LIN {X 0,Y 696.84,Z 1074.1,A -85,B 0,C 180,E1 3614.763,E2 3614.763} C_VEL
LIN {X 0,Y 697.033,Z 1060.691,A -85,B 0,C 180,E1 3616.923,E2 3616.923} C_VEL
LIN {X 0,Y 697.324,Z 1042.875,A -85,B 0,C 180,E1 3618.806,E2 3618.806} C_VEL
LIN {X 0,Y 697.62,Z 1019.345,A -85,B 0,C 180,E1 3620.491,E2 3620.491} C_VEL
LIN {X 0,Y 698.013,Z 992.248,A -85,B 0,C 180,E1 3621.752,E2 3621.752} C_VEL
LIN {X 0,Y 698.325,Z 962.562,A -85,B 0,C 180,E1 3622.528,E2 3622.528} C_VEL
LIN {X 0,Y 697.391,Z 928.875,A -85,B 0,C 180,E1 3622.939,E2 3622.939} C_VEL
LIN {X 0,Y 696.362,Z 923.03,A -85,B 0,C 180,E1 3623.04,E2 3623.04} C_VEL
LIN {X 0,Y 696.127,Z 923.03,A -85,B 0,C 180,E1 3627.121,E2 3627.121} C_VEL
LIN {X 0,Y 696.052,Z 923.03,A -85,B 0,C 180,E1 3632.136,E2 3632.136} C_VEL
LIN {X 0,Y 696.075,Z 923.03,A -85,B 0,C 180,E1 3637.436,E2 3637.436} C_VEL
LIN {X 0,Y 695.88,Z 923.03,A -85,B 0,C 180,E1 3642.402,E2 3642.402} C_VEL
LIN {X 0,Y 696.007,Z 923.03,A -85,B 0,C 180,E1 3647.688,E2 3647.688} C_VEL
LIN {X 0,Y 696.066,Z 923.03,A -85,B 0,C 180,E1 3652.556,E2 3652.556} C_VEL
LIN {X 0,Y 696.017,Z 923.03,A -85,B 0,C 180,E1 3657.859,E2 3657.859} C_VEL
LIN {X 0,Y 696.298,Z 923.03,A -85,B 0,C 180,E1 3662.878,E2 3662.878} C_VEL
LIN {X 0,Y 696.247,Z 923.03,A -85,B 0,C 180,E1 3668.339,E2 3668.339} C_VEL
LIN {X 0,Y 696.266,Z 923.03,A -85,B 0,C 180,E1 3673.602,E2 3673.602} C_VEL
LIN {X 0,Y 696.358,Z 923.03,A -85,B 0,C 180,E1 3678.728,E2 3678.728} C_VEL
LIN {X 0,Y 696.496,Z 923.03,A -85,B 0,C 180,E1 3683.762,E2 3683.762} C_VEL
LIN {X 0,Y 696.447,Z 923.03,A -85,B 0,C 180,E1 3688.746,E2 3688.746} C_VEL
LIN {X 0,Y 696.437,Z 923.03,A -85,B 0,C 180,E1 3692.476,E2 3692.476} C_VEL
LIN {X 0,Y 696.418,Z 923.03,A -85,B 0,C 180,E1 3696.217,E2 3696.217} C_VEL
LIN {X 0,Y 696.336,Z 923.03,A -85,B 0,C 180,E1 3701.25,E2 3701.25} C_VEL
LIN {X 0,Y 696.388,Z 923.03,A -85,B 0,C 180,E1 3706.372,E2 3706.372} C_VEL
LIN {X 0,Y 696.229,Z 923.03,A -85,B 0,C 180,E1 3711.638,E2 3711.638} C_VEL
LIN {X 0,Y 696.274,Z 923.03,A -85,B 0,C 180,E1 3715.71,E2 3715.71} C_VEL
LIN {X 0,Y 696.189,Z 923.03,A -85,B 0,C 180,E1 3719.933,E2 3719.933} C_VEL
LIN {X 0,Y 696.124,Z 923.03,A -85,B 0,C 180,E1 3724.422,E2 3724.422} C_VEL
LIN {X 0,Y 696.016,Z 923.03,A -85,B 0,C 180,E1 3729.003,E2 3729.003} C_VEL
LIN {X 0,Y 696.257,Z 923.03,A -85,B 0,C 180,E1 3734.256,E2 3734.256} C_VEL
LIN {X 0,Y 696.094,Z 923.03,A -85,B 0,C 180,E1 3739.422,E2 3739.422} C_VEL
LIN {X 0,Y 696.038,Z 923.03,A -85,B 0,C 180,E1 3744.113,E2 3744.113} C_VEL
LIN {X 0,Y 696.066,Z 923.03,A -85,B 0,C 180,E1 3748.598,E2 3748.598} C_VEL
LIN {X 0,Y 696.27,Z 923.03,A -85,B 0,C 180,E1 3752.885,E2 3752.885} C_VEL
LIN {X 0,Y 696.419,Z 923.03,A -85,B 0,C 180,E1 3755.045,E2 3755.045} C_VEL
LIN {X 0,Y 702.161,Z 942.704,A -85,B 0,C 180,E1 3755.601,E2 3755.601} C_VEL
LIN {X 0,Y 701.459,Z 983.403,A -85,B 0,C 180,E1 3756.655,E2 3756.655} C_VEL
LIN {X 0,Y 700.459,Z 1020.42,A -85,B 0,C 180,E1 3758.118,E2 3758.118} C_VEL
LIN {X 0,Y 699.341,Z 1055.77,A -85,B 0,C 180,E1 3760.059,E2 3760.059} C_VEL
LIN {X 0,Y 698.44,Z 1087.21,A -85,B 0,C 180,E1 3762.367,E2 3762.367} C_VEL
LIN {X 0,Y 697.692,Z 1115.392,A -85,B 0,C 180,E1 3765.095,E2 3765.095} C_VEL
LIN {X 0,Y 697.113,Z 1138.714,A -85,B 0,C 180,E1 3768.115,E2 3768.115} C_VEL
LIN {X 0,Y 696.808,Z 1156.179,A -85,B 0,C 180,E1 3771.267,E2 3771.267} C_VEL
LIN {X 0,Y 696.688,Z 1167.713,A -85,B 0,C 180,E1 3774.397,E2 3774.397} C_VEL
LIN {X 0,Y 696.627,Z 1173.967,A -85,B 0,C 180,E1 3777.512,E2 3777.512} C_VEL
LIN {X 0,Y 696.49,Z 1175.495,A -85,B 0,C 180,E1 3779.999,E2 3779.999} C_VEL
LIN {X 0,Y 696.656,Z 1173.847,A -85,B 0,C 180,E1 3782.485,E2 3782.485} C_VEL
LIN {X 0,Y 696.704,Z 1167.444,A -85,B 0,C 180,E1 3785.6,E2 3785.6} C_VEL
LIN {X 0,Y 696.77,Z 1155.784,A -85,B 0,C 180,E1 3788.73,E2 3788.73} C_VEL
LIN {X 0,Y 697.098,Z 1138.122,A -85,B 0,C 180,E1 3791.883,E2 3791.883} C_VEL
LIN {X 0,Y 697.634,Z 1114.595,A -85,B 0,C 180,E1 3794.904,E2 3794.904} C_VEL
LIN {X 0,Y 697.968,Z 1103.957,A -85,B 0,C 180,E1 3796.014,E2 3796.014} C_VEL
LIN {X 0,Y 694.387,Z 1093.241,A -85,B 0,C 180,E1 3797.118,E2 3797.118} C_VEL
LIN {X 0,Y 690.934,Z 1081.896,A -85,B 0,C 180,E1 3798.188,E2 3798.188} C_VEL
LIN {X 0,Y 692.119,Z 1048.543,A -85,B 0,C 180,E1 3800.528,E2 3800.528} C_VEL
LIN {X 0,Y 693.322,Z 1012.284,A -85,B 0,C 180,E1 3802.409,E2 3802.409} C_VEL
LIN {X 0,Y 694.361,Z 974.431,A -85,B 0,C 180,E1 3803.796,E2 3803.796} C_VEL
LIN {X 0,Y 694.245,Z 940.568,A -85,B 0,C 180,E1 3804.648,E2 3804.648} C_VEL
LIN {X 0,Y 688.268,Z 923.03,A -85,B 0,C 180,E1 3805.177,E2 3805.177} C_VEL
LIN {X 0,Y 688.234,Z 923.03,A -85,B 0,C 180,E1 3810.329,E2 3810.329} C_VEL
LIN {X 0,Y 688.148,Z 923.03,A -85,B 0,C 180,E1 3815.688,E2 3815.688} C_VEL
LIN {X 0,Y 688.036,Z 923.03,A -85,B 0,C 180,E1 3821.212,E2 3821.212} C_VEL
LIN {X 0,Y 688.049,Z 923.03,A -85,B 0,C 180,E1 3826.446,E2 3826.446} C_VEL
LIN {X 0,Y 688.208,Z 923.03,A -85,B 0,C 180,E1 3832.225,E2 3832.225} C_VEL
LIN {X 0,Y 688.212,Z 923.03,A -85,B 0,C 180,E1 3836.724,E2 3836.724} C_VEL
LIN {X 0,Y 688.234,Z 923.03,A -85,B 0,C 180,E1 3841.429,E2 3841.429} C_VEL
LIN {X 0,Y 688.093,Z 923.327,A -85,B 0,C 180,E1 3844.092,E2 3844.092} C_VEL
LIN {X 0,Y 695.508,Z 945.947,A -85,B 0,C 180,E1 3844.641,E2 3844.641} C_VEL
LIN {X 0,Y 695.052,Z 1003.247,A -85,B 0,C 180,E1 3845.392,E2 3845.392} C_VEL
LIN {X 0,Y 694.208,Z 1042.654,A -85,B 0,C 180,E1 3846.416,E2 3846.416} C_VEL
LIN {X 0,Y 693.113,Z 1079.521,A -85,B 0,C 180,E1 3847.875,E2 3847.875} C_VEL
LIN {X 0,Y 691.948,Z 1114.634,A -85,B 0,C 180,E1 3849.81,E2 3849.81} C_VEL
LIN {X 0,Y 690.803,Z 1145.44,A -85,B 0,C 180,E1 3852.063,E2 3852.063} C_VEL
LIN {X 0,Y 689.951,Z 1172.229,A -85,B 0,C 180,E1 3854.62,E2 3854.62} C_VEL
LIN {X 0,Y 689.296,Z 1195.231,A -85,B 0,C 180,E1 3857.51,E2 3857.51} C_VEL
LIN {X 0,Y 688.941,Z 1212.25,A -85,B 0,C 180,E1 3860.393,E2 3860.393} C_VEL
LIN {X 0,Y 688.809,Z 1224.727,A -85,B 0,C 180,E1 3863.398,E2 3863.398} C_VEL
LIN {X 0,Y 688.734,Z 1231.97,A -85,B 0,C 180,E1 3866.237,E2 3866.237} C_VEL
LIN {X 0,Y 688.725,Z 1235.095,A -85,B 0,C 180,E1 3868.754,E2 3868.754} C_VEL
LIN {X 0,Y 688.851,Z 1235.078,A -85,B 0,C 180,E1 3871.268,E2 3871.268} C_VEL
LIN {X 0,Y 688.802,Z 1230.721,A -85,B 0,C 180,E1 3874.414,E2 3874.414} C_VEL
LIN {X 0,Y 688.94,Z 1219.976,A -85,B 0,C 180,E1 3877.89,E2 3877.89} C_VEL
LIN {X 0,Y 689.179,Z 1204.28,A -85,B 0,C 180,E1 3881.071,E2 3881.071} C_VEL
LIN {X 0,Y 689.655,Z 1183.093,A -85,B 0,C 180,E1 3884.119,E2 3884.119} C_VEL
LIN {X 0,Y 690.437,Z 1157.494,A -85,B 0,C 180,E1 3886.867,E2 3886.867} C_VEL
LIN {X 0,Y 691.422,Z 1128.305,A -85,B 0,C 180,E1 3889.265,E2 3889.265} C_VEL
LIN {X 0,Y 692.587,Z 1094.665,A -85,B 0,C 180,E1 3891.361,E2 3891.361} C_VEL
LIN {X 0,Y 693.775,Z 1058.061,A -85,B 0,C 180,E1 3893.036,E2 3893.036} C_VEL
LIN {X 0,Y 694.758,Z 1021.242,A -85,B 0,C 180,E1 3894.199,E2 3894.199} C_VEL
LIN {X 0,Y 695.371,Z 982.472,A -85,B 0,C 180,E1 3894.941,E2 3894.941} C_VEL
LIN {X 0,Y 694.761,Z 941.711,A -85,B 0,C 180,E1 3895.435,E2 3895.435} C_VEL
LIN {X 0,Y 688.099,Z 923.03,A -85,B 0,C 180,E1 3895.984,E2 3895.984} C_VEL
LIN {X 0,Y 688.244,Z 923.03,A -85,B 0,C 180,E1 3901.101,E2 3901.101} C_VEL
LIN {X 0,Y 688.201,Z 923.03,A -85,B 0,C 180,E1 3906.369,E2 3906.369} C_VEL
LIN {X 0,Y 688.063,Z 923.03,A -85,B 0,C 180,E1 3911.697,E2 3911.697} C_VEL
LIN {X 0,Y 688.076,Z 923.03,A -85,B 0,C 180,E1 3917.096,E2 3917.096} C_VEL
LIN {X 0,Y 688.182,Z 923.03,A -85,B 0,C 180,E1 3922.242,E2 3922.242} C_VEL
LIN {X 0,Y 688.174,Z 923.03,A -85,B 0,C 180,E1 3926.707,E2 3926.707} C_VEL
LIN {X 0,Y 688.271,Z 923.03,A -85,B 0,C 180,E1 3931.439,E2 3931.439} C_VEL
LIN {X 0,Y 688.328,Z 923.03,A -85,B 0,C 180,E1 3936.726,E2 3936.726} C_VEL
LIN {X 0,Y 688.194,Z 923.03,A -85,B 0,C 180,E1 3940.782,E2 3940.782} C_VEL
LIN {X 0,Y 688.276,Z 923.03,A -85,B 0,C 180,E1 3946.026,E2 3946.026} C_VEL
LIN {X 0,Y 688.465,Z 923.03,A -85,B 0,C 180,E1 3951.163,E2 3951.163} C_VEL
LIN {X 0,Y 688.379,Z 923.03,A -85,B 0,C 180,E1 3956.225,E2 3956.225} C_VEL
LIN {X 0,Y 688.46,Z 923.03,A -85,B 0,C 180,E1 3956.751,E2 3956.751} C_VEL
LIN {X 0,Y 690.605,Z 940.887,A -85,B 0,C 180,E1 3956.98,E2 3956.98} C_VEL
LIN {X 0,Y 690.561,Z 973.087,A -85,B 0,C 180,E1 3957.459,E2 3957.459} C_VEL
LIN {X 0,Y 690.211,Z 1001.252,A -85,B 0,C 180,E1 3958.355,E2 3958.355} C_VEL
LIN {X 0,Y 689.834,Z 1026.543,A -85,B 0,C 180,E1 3959.688,E2 3959.688} C_VEL
LIN {X 0,Y 689.487,Z 1048.295,A -85,B 0,C 180,E1 3961.414,E2 3961.414} C_VEL
LIN {X 0,Y 689.207,Z 1065.525,A -85,B 0,C 180,E1 3963.458,E2 3963.458} C_VEL
LIN {X 0,Y 688.957,Z 1077.507,A -85,B 0,C 180,E1 3965.666,E2 3965.666} C_VEL
LIN {X 0,Y 688.864,Z 1084.771,A -85,B 0,C 180,E1 3968.199,E2 3968.199} C_VEL
LIN {X 0,Y 688.818,Z 1086.093,A -85,B 0,C 180,E1 3970.109,E2 3970.109} C_VEL
LIN {X 0,Y 688.951,Z 1082.737,A -85,B 0,C 180,E1 3972.671,E2 3972.671} C_VEL
LIN {X 0,Y 689.052,Z 1074.592,A -85,B 0,C 180,E1 3974.891,E2 3974.891} C_VEL
LIN {X 0,Y 689.218,Z 1060.902,A -85,B 0,C 180,E1 3977.073,E2 3977.073} C_VEL
LIN {X 0,Y 689.561,Z 1042.201,A -85,B 0,C 180,E1 3979.026,E2 3979.026} C_VEL
LIN {X 0,Y 689.91,Z 1019.357,A -85,B 0,C 180,E1 3980.646,E2 3980.646} C_VEL
LIN {X 0,Y 690.313,Z 992.621,A -85,B 0,C 180,E1 3981.886,E2 3981.886} C_VEL
LIN {X 0,Y 690.598,Z 964.533,A -85,B 0,C 180,E1 3982.633,E2 3982.633} C_VEL
LIN {X 0,Y 689.84,Z 930.872,A -85,B 0,C 180,E1 3983.057,E2 3983.057} C_VEL
LIN {X 0,Y 688.486,Z 923.03,A -85,B 0,C 180,E1 3983.204,E2 3983.204} C_VEL
LIN {X 0,Y 688.186,Z 923.03,A -85,B 0,C 180,E1 3988.548,E2 3988.548} C_VEL
LIN {X 0,Y 688.138,Z 923.03,A -85,B 0,C 180,E1 3993.429,E2 3993.429} C_VEL
LIN {X 0,Y 688.161,Z 923.03,A -85,B 0,C 180,E1 3997.942,E2 3997.942} C_VEL
LIN {X 0,Y 688.005,Z 923.03,A -85,B 0,C 180,E1 4003.538,E2 4003.538} C_VEL
LIN {X 0,Y 688.091,Z 923.03,A -85,B 0,C 180,E1 4008.78,E2 4008.78} C_VEL
LIN {X 0,Y 688.117,Z 923.03,A -85,B 0,C 180,E1 4013.626,E2 4013.626} C_VEL
LIN {X 0,Y 688.131,Z 923.03,A -85,B 0,C 180,E1 4018.919,E2 4018.919} C_VEL
LIN {X 0,Y 688.444,Z 923.03,A -85,B 0,C 180,E1 4024.152,E2 4024.152} C_VEL
LIN {X 0,Y 688.312,Z 923.03,A -85,B 0,C 180,E1 4029.426,E2 4029.426} C_VEL
LIN {X 0,Y 688.395,Z 923.03,A -85,B 0,C 180,E1 4034.717,E2 4034.717} C_VEL
LIN {X 0,Y 688.52,Z 923.03,A -85,B 0,C 180,E1 4039.878,E2 4039.878} C_VEL
LIN {X 0,Y 688.527,Z 923.03,A -85,B 0,C 180,E1 4044.953,E2 4044.953} C_VEL
LIN {X 0,Y 688.624,Z 923.03,A -85,B 0,C 180,E1 4049.989,E2 4049.989} C_VEL
LIN {X 0,Y 688.687,Z 923.03,A -85,B 0,C 180,E1 4055.024,E2 4055.024} C_VEL
LIN {X 0,Y 688.471,Z 923.03,A -85,B 0,C 180,E1 4060.101,E2 4060.101} C_VEL
LIN {X 0,Y 688.446,Z 923.03,A -85,B 0,C 180,E1 4065.259,E2 4065.259} C_VEL
LIN {X 0,Y 688.35,Z 923.03,A -85,B 0,C 180,E1 4070.549,E2 4070.549} C_VEL
LIN {X 0,Y 688.337,Z 923.03,A -85,B 0,C 180,E1 4076.029,E2 4076.029} C_VEL
LIN {X 0,Y 688.237,Z 923.03,A -85,B 0,C 180,E1 4081.095,E2 4081.095} C_VEL
LIN {X 0,Y 688.154,Z 923.03,A -85,B 0,C 180,E1 4086.344,E2 4086.344} C_VEL
LIN {X 0,Y 688.212,Z 923.03,A -85,B 0,C 180,E1 4091.707,E2 4091.707} C_VEL
LIN {X 0,Y 688.162,Z 923.03,A -85,B 0,C 180,E1 4096.416,E2 4096.416} C_VEL
LIN {X 0,Y 688.155,Z 923.03,A -85,B 0,C 180,E1 4102.208,E2 4102.208} C_VEL
LIN {X 0,Y 688.081,Z 923.03,A -85,B 0,C 180,E1 4106.698,E2 4106.698} C_VEL
LIN {X 0,Y 688.281,Z 923.03,A -85,B 0,C 180,E1 4111.391,E2 4111.391} C_VEL
LIN {X 0,Y 688.51,Z 923.03,A -85,B 0,C 180,E1 4114.742,E2 4114.742} C_VEL
LIN {X 0,Y 694.954,Z 944.35,A -85,B 0,C 180,E1 4115.367,E2 4115.367} C_VEL
LIN {X 0,Y 694.144,Z 984.038,A -85,B 0,C 180,E1 4116.417,E2 4116.417} C_VEL
LIN {X 0,Y 693.005,Z 1021.584,A -85,B 0,C 180,E1 4117.928,E2 4117.928} C_VEL
LIN {X 0,Y 691.779,Z 1056.552,A -85,B 0,C 180,E1 4119.884,E2 4119.884} C_VEL
LIN {X 0,Y 690.716,Z 1089.12,A -85,B 0,C 180,E1 4122.328,E2 4122.328} C_VEL
LIN {X 0,Y 689.888,Z 1116.828,A -85,B 0,C 180,E1 4125.085,E2 4125.085} C_VEL
LIN {X 0,Y 689.277,Z 1138.709,A -85,B 0,C 180,E1 4127.978,E2 4127.978} C_VEL
LIN {X 0,Y 688.922,Z 1156.175,A -85,B 0,C 180,E1 4131.167,E2 4131.167} C_VEL
LIN {X 0,Y 688.798,Z 1167.714,A -85,B 0,C 180,E1 4134.333,E2 4134.333} C_VEL
LIN {X 0,Y 688.737,Z 1173.968,A -85,B 0,C 180,E1 4137.484,E2 4137.484} C_VEL
LIN {X 0,Y 688.607,Z 1175.495,A -85,B 0,C 180,E1 4139.999,E2 4139.999} C_VEL
LIN {X 0,Y 688.764,Z 1173.849,A -85,B 0,C 180,E1 4142.514,E2 4142.514} C_VEL
LIN {X 0,Y 688.824,Z 1167.447,A -85,B 0,C 180,E1 4145.664,E2 4145.664} C_VEL
LIN {X 0,Y 688.893,Z 1155.788,A -85,B 0,C 180,E1 4148.831,E2 4148.831} C_VEL
LIN {X 0,Y 689.267,Z 1138.128,A -85,B 0,C 180,E1 4152.02,E2 4152.02} C_VEL
LIN {X 0,Y 689.873,Z 1114.603,A -85,B 0,C 180,E1 4155.075,E2 4155.075} C_VEL
LIN {X 0,Y 690.742,Z 1086.176,A -85,B 0,C 180,E1 4157.833,E2 4157.833} C_VEL
LIN {X 0,Y 690.934,Z 1081.896,A -85,B 0,C 180,E1 4158.188,E2 4158.188} C_VEL
LIN {X 0,Y 687.679,Z 1069.975,A -85,B 0,C 180,E1 4159.221,E2 4159.221} C_VEL
LIN {X 0,Y 684.251,Z 1057.373,A -85,B 0,C 180,E1 4160.202,E2 4160.202} C_VEL
LIN {X 0,Y 685.644,Z 1021.898,A -85,B 0,C 180,E1 4162.215,E2 4162.215} C_VEL
LIN {X 0,Y 686.89,Z 985.188,A -85,B 0,C 180,E1 4163.716,E2 4163.716} C_VEL
LIN {X 0,Y 687.745,Z 947.019,A -85,B 0,C 180,E1 4164.76,E2 4164.76} C_VEL
LIN {X 0,Y 680.378,Z 923.03,A -85,B 0,C 180,E1 4165.492,E2 4165.492} C_VEL
LIN {X 0,Y 680.326,Z 923.03,A -85,B 0,C 180,E1 4170.72,E2 4170.72} C_VEL
LIN {X 0,Y 680.25,Z 923.03,A -85,B 0,C 180,E1 4175.277,E2 4175.277} C_VEL
LIN {X 0,Y 680.106,Z 923.03,A -85,B 0,C 180,E1 4180.96,E2 4180.96} C_VEL
LIN {X 0,Y 680.126,Z 923.03,A -85,B 0,C 180,E1 4185.312,E2 4185.312} C_VEL
LIN {X 0,Y 680.126,Z 923.03,A -85,B 0,C 180,E1 4189.905,E2 4189.905} C_VEL
LIN {X 0,Y 680.338,Z 923.03,A -85,B 0,C 180,E1 4195.264,E2 4195.264} C_VEL
LIN {X 0,Y 680.244,Z 923.03,A -85,B 0,C 180,E1 4200.76,E2 4200.76} C_VEL
LIN {X 0,Y 680.16,Z 923.03,A -85,B 0,C 180,E1 4203.741,E2 4203.741} C_VEL
LIN {X 0,Y 688.35,Z 947.087,A -85,B 0,C 180,E1 4204.372,E2 4204.372} C_VEL
LIN {X 0,Y 687.847,Z 1003.636,A -85,B 0,C 180,E1 4205.125,E2 4205.125} C_VEL
LIN {X 0,Y 686.915,Z 1043.264,A -85,B 0,C 180,E1 4206.171,E2 4206.171} C_VEL
LIN {X 0,Y 685.661,Z 1080.997,A -85,B 0,C 180,E1 4207.696,E2 4207.696} C_VEL
LIN {X 0,Y 684.358,Z 1116.077,A -85,B 0,C 180,E1 4209.673,E2 4209.673} C_VEL
LIN {X 0,Y 683.069,Z 1147.5,A -85,B 0,C 180,E1 4212.032,E2 4212.032} C_VEL
LIN {X 0,Y 682.145,Z 1173.624,A -85,B 0,C 180,E1 4214.597,E2 4214.597} C_VEL
LIN {X 0,Y 681.505,Z 1194.886,A -85,B 0,C 180,E1 4217.313,E2 4217.313} C_VEL
LIN {X 0,Y 681.089,Z 1211.899,A -85,B 0,C 180,E1 4220.207,E2 4220.207} C_VEL
LIN {X 0,Y 680.936,Z 1224.727,A -85,B 0,C 180,E1 4223.321,E2 4223.321} C_VEL
LIN {X 0,Y 680.859,Z 1231.971,A -85,B 0,C 180,E1 4226.194,E2 4226.194} C_VEL
LIN {X 0,Y 680.825,Z 1235.095,A -85,B 0,C 180,E1 4228.74,E2 4228.74} C_VEL
LIN {X 0,Y 680.949,Z 1235.078,A -85,B 0,C 180,E1 4231.283,E2 4231.283} C_VEL
LIN {X 0,Y 680.912,Z 1230.721,A -85,B 0,C 180,E1 4234.466,E2 4234.466} C_VEL
LIN {X 0,Y 681.074,Z 1219.977,A -85,B 0,C 180,E1 4237.981,E2 4237.981} C_VEL
LIN {X 0,Y 681.332,Z 1204.279,A -85,B 0,C 180,E1 4241.2,E2 4241.2} C_VEL
LIN {X 0,Y 681.869,Z 1183.091,A -85,B 0,C 180,E1 4244.283,E2 4244.283} C_VEL
LIN {X 0,Y 682.729,Z 1157.713,A -85,B 0,C 180,E1 4247.043,E2 4247.043} C_VEL
LIN {X 0,Y 683.848,Z 1128.546,A -85,B 0,C 180,E1 4249.469,E2 4249.469} C_VEL
LIN {X 0,Y 685.086,Z 1096.194,A -85,B 0,C 180,E1 4251.522,E2 4251.522} C_VEL
LIN {X 0,Y 686.395,Z 1059.716,A -85,B 0,C 180,E1 4253.231,E2 4253.231} C_VEL
LIN {X 0,Y 687.52,Z 1021.63,A -85,B 0,C 180,E1 4254.461,E2 4254.461} C_VEL
LIN {X 0,Y 688.199,Z 984.433,A -85,B 0,C 180,E1 4255.193,E2 4255.193} C_VEL
LIN {X 0,Y 687.932,Z 944.356,A -85,B 0,C 180,E1 4255.676,E2 4255.676} C_VEL
LIN {X 0,Y 680.205,Z 923.03,A -85,B 0,C 180,E1 4256.281,E2 4256.281} C_VEL
LIN {X 0,Y 680.323,Z 923.03,A -85,B 0,C 180,E1 4260.731,E2 4260.731} C_VEL
LIN {X 0,Y 680.297,Z 923.03,A -85,B 0,C 180,E1 4265.286,E2 4265.286} C_VEL
LIN {X 0,Y 680.12,Z 923.03,A -85,B 0,C 180,E1 4270.94,E2 4270.94} C_VEL
LIN {X 0,Y 680.166,Z 923.03,A -85,B 0,C 180,E1 4275.321,E2 4275.321} C_VEL
LIN {X 0,Y 680.107,Z 923.03,A -85,B 0,C 180,E1 4279.886,E2 4279.886} C_VEL
LIN {X 0,Y 680.326,Z 923.03,A -85,B 0,C 180,E1 4285.279,E2 4285.279} C_VEL
LIN {X 0,Y 680.266,Z 923.03,A -85,B 0,C 180,E1 4290.747,E2 4290.747} C_VEL
LIN {X 0,Y 680.408,Z 923.03,A -85,B 0,C 180,E1 4295.598,E2 4295.598} C_VEL
LIN {X 0,Y 680.292,Z 923.03,A -85,B 0,C 180,E1 4300.539,E2 4300.539} C_VEL
LIN {X 0,Y 680.376,Z 923.03,A -85,B 0,C 180,E1 4305.861,E2 4305.861} C_VEL
LIN {X 0,Y 680.564,Z 923.03,A -85,B 0,C 180,E1 4311.06,E2 4311.06} C_VEL
LIN {X 0,Y 680.474,Z 923.03,A -85,B 0,C 180,E1 4316.182,E2 4316.182} C_VEL
LIN {X 0,Y 680.564,Z 923.609,A -85,B 0,C 180,E1 4316.613,E2 4316.613} C_VEL
LIN {X 0,Y 682.88,Z 942.51,A -85,B 0,C 180,E1 4316.858,E2 4316.858} C_VEL
LIN {X 0,Y 682.841,Z 974.882,A -85,B 0,C 180,E1 4317.356,E2 4317.356} C_VEL
LIN {X 0,Y 682.452,Z 1004.475,A -85,B 0,C 180,E1 4318.336,E2 4318.336} C_VEL
LIN {X 0,Y 682.039,Z 1030.175,A -85,B 0,C 180,E1 4319.763,E2 4319.763} C_VEL
LIN {X 0,Y 681.666,Z 1051.792,A -85,B 0,C 180,E1 4321.589,E2 4321.589} C_VEL
LIN {X 0,Y 681.384,Z 1067.669,A -85,B 0,C 180,E1 4323.568,E2 4323.568} C_VEL
LIN {X 0,Y 681.135,Z 1078.931,A -85,B 0,C 180,E1 4325.731,E2 4325.731} C_VEL
LIN {X 0,Y 681.042,Z 1084.694,A -85,B 0,C 180,E1 4327.652,E2 4327.652} C_VEL
LIN {X 0,Y 680.984,Z 1087.044,A -85,B 0,C 180,E1 4330.227,E2 4330.227} C_VEL
LIN {X 0,Y 681.102,Z 1084.11,A -85,B 0,C 180,E1 4332.501,E2 4332.501} C_VEL
LIN {X 0,Y 681.204,Z 1076.61,A -85,B 0,C 180,E1 4334.696,E2 4334.696} C_VEL
LIN {X 0,Y 681.445,Z 1063.248,A -85,B 0,C 180,E1 4336.952,E2 4336.952} C_VEL
LIN {X 0,Y 681.779,Z 1045.397,A -85,B 0,C 180,E1 4338.915,E2 4338.915} C_VEL
LIN {X 0,Y 682.116,Z 1022.099,A -85,B 0,C 180,E1 4340.641,E2 4340.641} C_VEL
LIN {X 0,Y 682.577,Z 995.081,A -85,B 0,C 180,E1 4341.946,E2 4341.946} C_VEL
LIN {X 0,Y 682.892,Z 966.819,A -85,B 0,C 180,E1 4342.735,E2 4342.735} C_VEL
LIN {X 0,Y 681.874,Z 930.202,A -85,B 0,C 180,E1 4343.212,E2 4343.212} C_VEL
LIN {X 0,Y 680.564,Z 923.03,A -85,B 0,C 180,E1 4343.386,E2 4343.386} C_VEL
LIN {X 0,Y 680.266,Z 923.03,A -85,B 0,C 180,E1 4347.808,E2 4347.808} C_VEL
LIN {X 0,Y 680.188,Z 923.03,A -85,B 0,C 180,E1 4352.401,E2 4352.401} C_VEL
LIN {X 0,Y 680.215,Z 923.03,A -85,B 0,C 180,E1 4356.883,E2 4356.883} C_VEL
LIN {X 0,Y 680.077,Z 923.03,A -85,B 0,C 180,E1 4361.806,E2 4361.806} C_VEL
LIN {X 0,Y 680.154,Z 923.03,A -85,B 0,C 180,E1 4367.154,E2 4367.154} C_VEL
LIN {X 0,Y 680.204,Z 923.03,A -85,B 0,C 180,E1 4371.525,E2 4371.525} C_VEL
LIN {X 0,Y 680.178,Z 923.03,A -85,B 0,C 180,E1 4376.251,E2 4376.251} C_VEL
LIN {X 0,Y 680.293,Z 923.03,A -85,B 0,C 180,E1 4380.737,E2 4380.737} C_VEL
LIN {X 0,Y 680.417,Z 923.03,A -85,B 0,C 180,E1 4385.584,E2 4385.584} C_VEL
LIN {X 0,Y 680.447,Z 923.03,A -85,B 0,C 180,E1 4390.532,E2 4390.532} C_VEL
LIN {X 0,Y 680.401,Z 923.03,A -85,B 0,C 180,E1 4395.849,E2 4395.849} C_VEL
LIN {X 0,Y 680.567,Z 923.03,A -85,B 0,C 180,E1 4401.048,E2 4401.048} C_VEL
LIN {X 0,Y 680.735,Z 923.03,A -85,B 0,C 180,E1 4406.171,E2 4406.171} C_VEL
LIN {X 0,Y 680.875,Z 923.03,A -85,B 0,C 180,E1 4411.26,E2 4411.26} C_VEL
LIN {X 0,Y 680.599,Z 923.03,A -85,B 0,C 180,E1 4416.362,E2 4416.362} C_VEL
LIN {X 0,Y 680.531,Z 923.03,A -85,B 0,C 180,E1 4421.515,E2 4421.515} C_VEL
LIN {X 0,Y 680.549,Z 923.03,A -85,B 0,C 180,E1 4426.764,E2 4426.764} C_VEL
LIN {X 0,Y 680.375,Z 923.03,A -85,B 0,C 180,E1 4432.169,E2 4432.169} C_VEL
LIN {X 0,Y 680.397,Z 923.03,A -85,B 0,C 180,E1 4437.329,E2 4437.329} C_VEL
LIN {X 0,Y 680.307,Z 923.03,A -85,B 0,C 180,E1 4442.427,E2 4442.427} C_VEL
LIN {X 0,Y 680.204,Z 923.03,A -85,B 0,C 180,E1 4446.891,E2 4446.891} C_VEL
LIN {X 0,Y 680.408,Z 923.03,A -85,B 0,C 180,E1 4452.869,E2 4452.869} C_VEL
LIN {X 0,Y 680.197,Z 923.03,A -85,B 0,C 180,E1 4458.203,E2 4458.203} C_VEL
LIN {X 0,Y 680.187,Z 923.03,A -85,B 0,C 180,E1 4463.141,E2 4463.141} C_VEL
LIN {X 0,Y 680.172,Z 923.03,A -85,B 0,C 180,E1 4467.777,E2 4467.777} C_VEL
LIN {X 0,Y 680.435,Z 923.03,A -85,B 0,C 180,E1 4472.627,E2 4472.627} C_VEL
LIN {X 0,Y 680.584,Z 923.03,A -85,B 0,C 180,E1 4474.438,E2 4474.438} C_VEL
LIN {X 0,Y 687.736,Z 947.024,A -85,B 0,C 180,E1 4475.151,E2 4475.151} C_VEL
LIN {X 0,Y 686.806,Z 986.299,A -85,B 0,C 180,E1 4476.23,E2 4476.23} C_VEL
LIN {X 0,Y 685.575,Z 1022.792,A -85,B 0,C 180,E1 4477.737,E2 4477.737} C_VEL
LIN {X 0,Y 684.164,Z 1058.764,A -85,B 0,C 180,E1 4479.798,E2 4479.798} C_VEL
LIN {X 0,Y 682.96,Z 1091.117,A -85,B 0,C 180,E1 4482.3,E2 4482.3} C_VEL
LIN {X 0,Y 682.063,Z 1118.176,A -85,B 0,C 180,E1 4485.074,E2 4485.074} C_VEL
LIN {X 0,Y 681.418,Z 1140.795,A -85,B 0,C 180,E1 4488.178,E2 4488.178} C_VEL
LIN {X 0,Y 681.055,Z 1157.532,A -85,B 0,C 180,E1 4491.385,E2 4491.385} C_VEL
LIN {X 0,Y 680.918,Z 1167.713,A -85,B 0,C 180,E1 4494.267,E2 4494.267} C_VEL
LIN {X 0,Y 680.834,Z 1173.968,A -85,B 0,C 180,E1 4497.454,E2 4497.454} C_VEL
LIN {X 0,Y 680.708,Z 1175.495,A -85,B 0,C 180,E1 4499.999,E2 4499.999} C_VEL
LIN {X 0,Y 680.838,Z 1173,A -85,B 0,C 180,E1 4503.168,E2 4503.168} C_VEL
LIN {X 0,Y 681.023,Z 1164.543,A -85,B 0,C 180,E1 4506.688,E2 4506.688} C_VEL
LIN {X 0,Y 681.142,Z 1151.421,A -85,B 0,C 180,E1 4509.843,E2 4509.843} C_VEL
LIN {X 0,Y 681.672,Z 1131.512,A -85,B 0,C 180,E1 4513.132,E2 4513.132} C_VEL
LIN {X 0,Y 682.431,Z 1106.593,A -85,B 0,C 180,E1 4516.12,E2 4516.12} C_VEL
LIN {X 0,Y 683.539,Z 1077.115,A -85,B 0,C 180,E1 4518.778,E2 4518.778} C_VEL
LIN {X 0,Y 684.251,Z 1057.373,A -85,B 0,C 180,E1 4520.202,E2 4520.202} C_VEL
LIN {X 0,Y 680.983,Z 1044.249,A -85,B 0,C 180,E1 4521.142,E2 4521.142} C_VEL
LIN {X 0,Y 677.931,Z 1032.438,A -85,B 0,C 180,E1 4521.927,E2 4521.927} C_VEL
LIN {X 0,Y 677.933,Z 1030.583,A -85,B 0,C 180,E1 4522.028,E2 4522.028} C_VEL
LIN {X 0,Y 679.33,Z 993.397,A -85,B 0,C 180,E1 4523.697,E2 4523.697} C_VEL
LIN {X 0,Y 680.46,Z 954.713,A -85,B 0,C 180,E1 4524.87,E2 4524.87} C_VEL
LIN {X 0,Y 679.739,Z 944.582,A -85,B 0,C 180,E1 4525.126,E2 4525.126} C_VEL
LIN {X 0,Y 672.425,Z 923.03,A -85,B 0,C 180,E1 4525.808,E2 4525.808} C_VEL
LIN {X 0,Y 672.394,Z 923.03,A -85,B 0,C 180,E1 4531.382,E2 4531.382} C_VEL
LIN {X 0,Y 672.277,Z 923.03,A -85,B 0,C 180,E1 4536.011,E2 4536.011} C_VEL
LIN {X 0,Y 672.2,Z 923.03,A -85,B 0,C 180,E1 4540.684,E2 4540.684} C_VEL
LIN {X 0,Y 672.21,Z 923.03,A -85,B 0,C 180,E1 4545.998,E2 4545.998} C_VEL
LIN {X 0,Y 672.264,Z 923.03,A -85,B 0,C 180,E1 4551.015,E2 4551.015} C_VEL
LIN {X 0,Y 672.432,Z 923.03,A -85,B 0,C 180,E1 4556.247,E2 4556.247} C_VEL
LIN {X 0,Y 672.3,Z 923.03,A -85,B 0,C 180,E1 4561.851,E2 4561.851} C_VEL
LIN {X 0,Y 672.26,Z 923.03,A -85,B 0,C 180,E1 4563.497,E2 4563.497} C_VEL
LIN {X 0,Y 681.08,Z 947.182,A -85,B 0,C 180,E1 4564.079,E2 4564.079} C_VEL
LIN {X 0,Y 680.703,Z 1003.108,A -85,B 0,C 180,E1 4564.834,E2 4564.834} C_VEL
LIN {X 0,Y 679.645,Z 1043.443,A -85,B 0,C 180,E1 4565.907,E2 4565.907} C_VEL
LIN {X 0,Y 678.304,Z 1080.37,A -85,B 0,C 180,E1 4567.409,E2 4567.409} C_VEL
LIN {X 0,Y 676.87,Z 1115.168,A -85,B 0,C 180,E1 4569.376,E2 4569.376} C_VEL
LIN {X 0,Y 675.445,Z 1146.806,A -85,B 0,C 180,E1 4571.761,E2 4571.761} C_VEL
LIN {X 0,Y 674.375,Z 1174.107,A -85,B 0,C 180,E1 4574.471,E2 4574.471} C_VEL
LIN {X 0,Y 673.674,Z 1195.795,A -85,B 0,C 180,E1 4577.301,E2 4577.301} C_VEL
LIN {X 0,Y 673.212,Z 1212.977,A -85,B 0,C 180,E1 4580.321,E2 4580.321} C_VEL
LIN {X 0,Y 673.029,Z 1225.69,A -85,B 0,C 180,E1 4583.566,E2 4583.566} C_VEL
LIN {X 0,Y 672.96,Z 1231.971,A -85,B 0,C 180,E1 4586.149,E2 4586.149} C_VEL
LIN {X 0,Y 672.93,Z 1235.096,A -85,B 0,C 180,E1 4588.725,E2 4588.725} C_VEL
LIN {X 0,Y 673.048,Z 1235.078,A -85,B 0,C 180,E1 4591.298,E2 4591.298} C_VEL
LIN {X 0,Y 673.022,Z 1230.721,A -85,B 0,C 180,E1 4594.518,E2 4594.518} C_VEL
LIN {X 0,Y 673.203,Z 1219.977,A -85,B 0,C 180,E1 4598.075,E2 4598.075} C_VEL
LIN {X 0,Y 673.487,Z 1204.278,A -85,B 0,C 180,E1 4601.332,E2 4601.332} C_VEL
LIN {X 0,Y 674.079,Z 1183.166,A -85,B 0,C 180,E1 4604.442,E2 4604.442} C_VEL
LIN {X 0,Y 675.035,Z 1158.061,A -85,B 0,C 180,E1 4607.21,E2 4607.21} C_VEL
LIN {X 0,Y 676.261,Z 1128.754,A -85,B 0,C 180,E1 4609.681,E2 4609.681} C_VEL
LIN {X 0,Y 677.662,Z 1096.19,A -85,B 0,C 180,E1 4611.77,E2 4611.77} C_VEL
LIN {X 0,Y 679.077,Z 1059.836,A -85,B 0,C 180,E1 4613.491,E2 4613.491} C_VEL
LIN {X 0,Y 680.313,Z 1021.667,A -85,B 0,C 180,E1 4614.736,E2 4614.736} C_VEL
LIN {X 0,Y 681.058,Z 984.433,A -85,B 0,C 180,E1 4615.476,E2 4615.476} C_VEL
LIN {X 0,Y 680.537,Z 945.557,A -85,B 0,C 180,E1 4615.962,E2 4615.962} C_VEL
LIN {X 0,Y 672.283,Z 923.03,A -85,B 0,C 180,E1 4616.574,E2 4616.574} C_VEL
LIN {X 0,Y 672.379,Z 923.03,A -85,B 0,C 180,E1 4621.352,E2 4621.352} C_VEL
LIN {X 0,Y 672.341,Z 923.03,A -85,B 0,C 180,E1 4625.994,E2 4625.994} C_VEL
LIN {X 0,Y 672.222,Z 923.03,A -85,B 0,C 180,E1 4630.695,E2 4630.695} C_VEL
LIN {X 0,Y 672.244,Z 923.03,A -85,B 0,C 180,E1 4636.008,E2 4636.008} C_VEL
LIN {X 0,Y 672.239,Z 923.03,A -85,B 0,C 180,E1 4640.996,E2 4640.996} C_VEL
LIN {X 0,Y 672.37,Z 923.03,A -85,B 0,C 180,E1 4646.27,E2 4646.27} C_VEL
LIN {X 0,Y 672.362,Z 923.03,A -85,B 0,C 180,E1 4651.84,E2 4651.84} C_VEL
LIN {X 0,Y 672.449,Z 923.03,A -85,B 0,C 180,E1 4657.138,E2 4657.138} C_VEL
LIN {X 0,Y 672.259,Z 923.03,A -85,B 0,C 180,E1 4661.659,E2 4661.659} C_VEL
LIN {X 0,Y 672.475,Z 923.03,A -85,B 0,C 180,E1 4667.016,E2 4667.016} C_VEL
LIN {X 0,Y 672.666,Z 923.03,A -85,B 0,C 180,E1 4671.315,E2 4671.315} C_VEL
LIN {X 0,Y 672.596,Z 923.03,A -85,B 0,C 180,E1 4676.438,E2 4676.438} C_VEL
LIN {X 0,Y 675.158,Z 942.54,A -85,B 0,C 180,E1 4676.716,E2 4676.716} C_VEL
LIN {X 0,Y 675.137,Z 975.276,A -85,B 0,C 180,E1 4677.216,E2 4677.216} C_VEL
LIN {X 0,Y 674.783,Z 1004.022,A -85,B 0,C 180,E1 4678.157,E2 4678.157} C_VEL
LIN {X 0,Y 674.318,Z 1030.224,A -85,B 0,C 180,E1 4679.6,E2 4679.6} C_VEL
LIN {X 0,Y 673.963,Z 1050.66,A -85,B 0,C 180,E1 4681.286,E2 4681.286} C_VEL
LIN {X 0,Y 673.622,Z 1067.725,A -85,B 0,C 180,E1 4683.363,E2 4683.363} C_VEL
LIN {X 0,Y 673.309,Z 1080.323,A -85,B 0,C 180,E1 4685.798,E2 4685.798} C_VEL
LIN {X 0,Y 673.207,Z 1085.886,A -85,B 0,C 180,E1 4687.741,E2 4687.741} C_VEL
LIN {X 0,Y 673.153,Z 1087.934,A -85,B 0,C 180,E1 4690.347,E2 4690.347} C_VEL
LIN {X 0,Y 673.268,Z 1085.047,A -85,B 0,C 180,E1 4692.511,E2 4692.511} C_VEL
LIN {X 0,Y 673.4,Z 1077.441,A -85,B 0,C 180,E1 4694.754,E2 4694.754} C_VEL
LIN {X 0,Y 673.639,Z 1063.348,A -85,B 0,C 180,E1 4697.127,E2 4697.127} C_VEL
LIN {X 0,Y 674.029,Z 1044.722,A -85,B 0,C 180,E1 4699.141,E2 4699.141} C_VEL
LIN {X 0,Y 674.413,Z 1021.791,A -85,B 0,C 180,E1 4700.82,E2 4700.82} C_VEL
LIN {X 0,Y 674.872,Z 995.46,A -85,B 0,C 180,E1 4702.086,E2 4702.086} C_VEL
LIN {X 0,Y 675.202,Z 967.093,A -85,B 0,C 180,E1 4702.876,E2 4702.876} C_VEL
LIN {X 0,Y 674.312,Z 931.967,A -85,B 0,C 180,E1 4703.337,E2 4703.337} C_VEL
LIN {X 0,Y 672.645,Z 923.03,A -85,B 0,C 180,E1 4703.507,E2 4703.507} C_VEL
LIN {X 0,Y 672.286,Z 923.03,A -85,B 0,C 180,E1 4708.751,E2 4708.751} C_VEL
LIN {X 0,Y 672.329,Z 923.03,A -85,B 0,C 180,E1 4714.188,E2 4714.188} C_VEL
LIN {X 0,Y 672.311,Z 923.03,A -85,B 0,C 180,E1 4719.003,E2 4719.003} C_VEL
LIN {X 0,Y 672.21,Z 923.03,A -85,B 0,C 180,E1 4724.178,E2 4724.178} C_VEL
LIN {X 0,Y 672.343,Z 923.03,A -85,B 0,C 180,E1 4729.834,E2 4729.834} C_VEL
LIN {X 0,Y 672.267,Z 923.03,A -85,B 0,C 180,E1 4734.228,E2 4734.228} C_VEL
LIN {X 0,Y 672.27,Z 923.03,A -85,B 0,C 180,E1 4738.86,E2 4738.86} C_VEL
LIN {X 0,Y 672.53,Z 923.03,A -85,B 0,C 180,E1 4743.998,E2 4743.998} C_VEL
LIN {X 0,Y 672.484,Z 923.03,A -85,B 0,C 180,E1 4748.919,E2 4748.919} C_VEL
LIN {X 0,Y 672.552,Z 923.03,A -85,B 0,C 180,E1 4754.348,E2 4754.348} C_VEL
LIN {X 0,Y 672.698,Z 923.03,A -85,B 0,C 180,E1 4759.637,E2 4759.637} C_VEL
LIN {X 0,Y 672.722,Z 923.03,A -85,B 0,C 180,E1 4764.834,E2 4764.834} C_VEL
LIN {X 0,Y 672.771,Z 923.03,A -85,B 0,C 180,E1 4768.702,E2 4768.702} C_VEL
LIN {X 0,Y 672.738,Z 923.03,A -85,B 0,C 180,E1 4772.563,E2 4772.563} C_VEL
LIN {X 0,Y 672.692,Z 923.03,A -85,B 0,C 180,E1 4776.437,E2 4776.437} C_VEL
LIN {X 0,Y 672.63,Z 923.03,A -85,B 0,C 180,E1 4781.652,E2 4781.652} C_VEL
LIN {X 0,Y 672.64,Z 923.03,A -85,B 0,C 180,E1 4786.967,E2 4786.967} C_VEL
LIN {X 0,Y 672.442,Z 923.03,A -85,B 0,C 180,E1 4792.444,E2 4792.444} C_VEL
LIN {X 0,Y 672.482,Z 923.03,A -85,B 0,C 180,E1 4796.69,E2 4796.69} C_VEL
LIN {X 0,Y 672.391,Z 923.03,A -85,B 0,C 180,E1 4801.349,E2 4801.349} C_VEL
LIN {X 0,Y 672.291,Z 923.03,A -85,B 0,C 180,E1 4805.983,E2 4805.983} C_VEL
LIN {X 0,Y 672.302,Z 923.03,A -85,B 0,C 180,E1 4810.659,E2 4810.659} C_VEL
LIN {X 0,Y 672.379,Z 923.03,A -85,B 0,C 180,E1 4815.836,E2 4815.836} C_VEL
LIN {X 0,Y 672.327,Z 923.03,A -85,B 0,C 180,E1 4820.998,E2 4820.998} C_VEL
LIN {X 0,Y 672.31,Z 923.03,A -85,B 0,C 180,E1 4826.237,E2 4826.237} C_VEL
LIN {X 0,Y 672.427,Z 923.03,A -85,B 0,C 180,E1 4831.84,E2 4831.84} C_VEL
LIN {X 0,Y 672.678,Z 923.03,A -85,B 0,C 180,E1 4834.134,E2 4834.134} C_VEL
LIN {X 0,Y 680.548,Z 947.85,A -85,B 0,C 180,E1 4834.889,E2 4834.889} C_VEL
LIN {X 0,Y 679.506,Z 986.482,A -85,B 0,C 180,E1 4835.965,E2 4835.965} C_VEL
LIN {X 0,Y 678.167,Z 1022.773,A -85,B 0,C 180,E1 4837.48,E2 4837.48} C_VEL
LIN {X 0,Y 676.741,Z 1057.595,A -85,B 0,C 180,E1 4839.488,E2 4839.488} C_VEL
LIN {X 0,Y 675.312,Z 1090.602,A -85,B 0,C 180,E1 4842.045,E2 4842.045} C_VEL
LIN {X 0,Y 674.31,Z 1118.168,A -85,B 0,C 180,E1 4844.898,E2 4844.898} C_VEL
LIN {X 0,Y 673.589,Z 1139.285,A -85,B 0,C 180,E1 4847.79,E2 4847.79} C_VEL
LIN {X 0,Y 673.2,Z 1156.167,A -85,B 0,C 180,E1 4850.959,E2 4850.959} C_VEL
LIN {X 0,Y 673.017,Z 1167.713,A -85,B 0,C 180,E1 4854.2,E2 4854.2} C_VEL
LIN {X 0,Y 672.949,Z 1173.968,A -85,B 0,C 180,E1 4857.425,E2 4857.425} C_VEL
LIN {X 0,Y 672.828,Z 1175.496,A -85,B 0,C 180,E1 4859.999,E2 4859.999} C_VEL
LIN {X 0,Y 672.974,Z 1173.852,A -85,B 0,C 180,E1 4862.573,E2 4862.573} C_VEL
LIN {X 0,Y 673.055,Z 1167.453,A -85,B 0,C 180,E1 4865.797,E2 4865.797} C_VEL
LIN {X 0,Y 673.169,Z 1155.488,A -85,B 0,C 180,E1 4869.105,E2 4869.105} C_VEL
LIN {X 0,Y 673.614,Z 1137.462,A -85,B 0,C 180,E1 4872.405,E2 4872.405} C_VEL
LIN {X 0,Y 674.435,Z 1114.123,A -85,B 0,C 180,E1 4875.485,E2 4875.485} C_VEL
LIN {X 0,Y 675.487,Z 1086.179,A -85,B 0,C 180,E1 4878.25,E2 4878.25} C_VEL
LIN {X 0,Y 676.866,Z 1054.118,A -85,B 0,C 180,E1 4880.649,E2 4880.649} C_VEL
LIN {X 0,Y 677.933,Z 1030.583,A -85,B 0,C 180,E1 4882.028,E2 4882.028} C_VEL
LIN {X 0,Y 674.947,Z 1016.459,A -85,B 0,C 180,E1 4882.871,E2 4882.871} C_VEL
LIN {X 0,Y 671.676,Z 1001.807,A -85,B 0,C 180,E1 4883.642,E2 4883.642} C_VEL
LIN {X 0,Y 672.981,Z 964.009,A -85,B 0,C 180,E1 4884.911,E2 4884.911} C_VEL
LIN {X 0,Y 672.55,Z 946.849,A -85,B 0,C 180,E1 4885.341,E2 4885.341} C_VEL
LIN {X 0,Y 664.501,Z 923.03,A -85,B 0,C 180,E1 4886.079,E2 4886.079} C_VEL
LIN {X 0,Y 664.505,Z 923.03,A -85,B 0,C 180,E1 4891.534,E2 4891.534} C_VEL
LIN {X 0,Y 664.365,Z 923.03,A -85,B 0,C 180,E1 4896.252,E2 4896.252} C_VEL
LIN {X 0,Y 664.277,Z 923.03,A -85,B 0,C 180,E1 4901.374,E2 4901.374} C_VEL
LIN {X 0,Y 664.277,Z 923.03,A -85,B 0,C 180,E1 4906.986,E2 4906.986} C_VEL
LIN {X 0,Y 664.428,Z 923.03,A -85,B 0,C 180,E1 4912.747,E2 4912.747} C_VEL
LIN {X 0,Y 664.453,Z 923.03,A -85,B 0,C 180,E1 4917.291,E2 4917.291} C_VEL
LIN {X 0,Y 664.334,Z 923.03,A -85,B 0,C 180,E1 4922.956,E2 4922.956} C_VEL
LIN {X 0,Y 664.364,Z 923.03,A -85,B 0,C 180,E1 4923.224,E2 4923.224} C_VEL
LIN {X 0,Y 673.855,Z 949.925,A -85,B 0,C 180,E1 4923.861,E2 4923.861} C_VEL
LIN {X 0,Y 673.445,Z 1003.513,A -85,B 0,C 180,E1 4924.575,E2 4924.575} C_VEL
LIN {X 0,Y 672.448,Z 1042.114,A -85,B 0,C 180,E1 4925.584,E2 4925.584} C_VEL
LIN {X 0,Y 670.912,Z 1080.479,A -85,B 0,C 180,E1 4927.152,E2 4927.152} C_VEL
LIN {X 0,Y 669.356,Z 1115.484,A -85,B 0,C 180,E1 4929.156,E2 4929.156} C_VEL
LIN {X 0,Y 667.828,Z 1146.805,A -85,B 0,C 180,E1 4931.546,E2 4931.546} C_VEL
LIN {X 0,Y 666.66,Z 1173.621,A -85,B 0,C 180,E1 4934.23,E2 4934.23} C_VEL
LIN {X 0,Y 665.848,Z 1196.228,A -85,B 0,C 180,E1 4937.216,E2 4937.216} C_VEL
LIN {X 0,Y 665.343,Z 1212.976,A -85,B 0,C 180,E1 4940.205,E2 4940.205} C_VEL
LIN {X 0,Y 665.135,Z 1225.689,A -85,B 0,C 180,E1 4943.49,E2 4943.49} C_VEL
LIN {X 0,Y 665.074,Z 1231.971,A -85,B 0,C 180,E1 4946.103,E2 4946.103} C_VEL
LIN {X 0,Y 665.035,Z 1235.096,A -85,B 0,C 180,E1 4948.71,E2 4948.71} C_VEL
LIN {X 0,Y 665.127,Z 1234.852,A -85,B 0,C 180,E1 4951.606,E2 4951.606} C_VEL
LIN {X 0,Y 665.167,Z 1229.181,A -85,B 0,C 180,E1 4955.225,E2 4955.225} C_VEL
LIN {X 0,Y 665.358,Z 1218.972,A -85,B 0,C 180,E1 4958.419,E2 4958.419} C_VEL
LIN {X 0,Y 665.65,Z 1204.277,A -85,B 0,C 180,E1 4961.468,E2 4961.468} C_VEL
LIN {X 0,Y 666.296,Z 1183.285,A -85,B 0,C 180,E1 4964.599,E2 4964.599} C_VEL
LIN {X 0,Y 667.357,Z 1157.26,A -85,B 0,C 180,E1 4967.492,E2 4967.492} C_VEL
LIN {X 0,Y 668.723,Z 1128.052,A -85,B 0,C 180,E1 4969.965,E2 4969.965} C_VEL
LIN {X 0,Y 670.258,Z 1094.904,A -85,B 0,C 180,E1 4972.096,E2 4972.096} C_VEL
LIN {X 0,Y 671.802,Z 1058.765,A -85,B 0,C 180,E1 4973.805,E2 4973.805} C_VEL
LIN {X 0,Y 673.101,Z 1022.11,A -85,B 0,C 180,E1 4975.001,E2 4975.001} C_VEL
LIN {X 0,Y 673.834,Z 983.813,A -85,B 0,C 180,E1 4975.757,E2 4975.757} C_VEL
LIN {X 0,Y 673.591,Z 948.229,A -85,B 0,C 180,E1 4976.193,E2 4976.193} C_VEL
LIN {X 0,Y 664.37,Z 923.03,A -85,B 0,C 180,E1 4976.854,E2 4976.854} C_VEL
LIN {X 0,Y 664.471,Z 923.03,A -85,B 0,C 180,E1 4981.547,E2 4981.547} C_VEL
LIN {X 0,Y 664.431,Z 923.03,A -85,B 0,C 180,E1 4986.26,E2 4986.26} C_VEL
LIN {X 0,Y 664.291,Z 923.03,A -85,B 0,C 180,E1 4991.354,E2 4991.354} C_VEL
LIN {X 0,Y 664.294,Z 923.03,A -85,B 0,C 180,E1 4996.969,E2 4996.969} C_VEL
LIN {X 0,Y 664.399,Z 923.03,A -85,B 0,C 180,E1 5002.765,E2 5002.765} C_VEL
LIN {X 0,Y 664.402,Z 923.03,A -85,B 0,C 180,E1 5007.314,E2 5007.314} C_VEL
LIN {X 0,Y 664.441,Z 923.03,A -85,B 0,C 180,E1 5012.946,E2 5012.946} C_VEL
LIN {X 0,Y 664.564,Z 923.03,A -85,B 0,C 180,E1 5017.262,E2 5017.262} C_VEL
LIN {X 0,Y 664.35,Z 923.03,A -85,B 0,C 180,E1 5022.802,E2 5022.802} C_VEL
LIN {X 0,Y 664.675,Z 923.03,A -85,B 0,C 180,E1 5028.195,E2 5028.195} C_VEL
LIN {X 0,Y 664.81,Z 923.03,A -85,B 0,C 180,E1 5033.476,E2 5033.476} C_VEL
LIN {X 0,Y 664.697,Z 923.03,A -85,B 0,C 180,E1 5036.28,E2 5036.28} C_VEL
LIN {X 0,Y 667.449,Z 943.479,A -85,B 0,C 180,E1 5036.58,E2 5036.58} C_VEL
LIN {X 0,Y 667.417,Z 976.912,A -85,B 0,C 180,E1 5037.103,E2 5037.103} C_VEL
LIN {X 0,Y 667.051,Z 1005.368,A -85,B 0,C 180,E1 5038.054,E2 5038.054} C_VEL
LIN {X 0,Y 666.58,Z 1031.468,A -85,B 0,C 180,E1 5039.514,E2 5039.514} C_VEL
LIN {X 0,Y 666.173,Z 1052.634,A -85,B 0,C 180,E1 5041.301,E2 5041.301} C_VEL
LIN {X 0,Y 665.811,Z 1069.668,A -85,B 0,C 180,E1 5043.449,E2 5043.449} C_VEL
LIN {X 0,Y 665.494,Z 1081.709,A -85,B 0,C 180,E1 5045.866,E2 5045.866} C_VEL
LIN {X 0,Y 665.381,Z 1087.04,A -85,B 0,C 180,E1 5047.833,E2 5047.833} C_VEL
LIN {X 0,Y 665.322,Z 1088.818,A -85,B 0,C 180,E1 5050.47,E2 5050.47} C_VEL
LIN {X 0,Y 665.439,Z 1086.198,A -85,B 0,C 180,E1 5052.429,E2 5052.429} C_VEL
LIN {X 0,Y 665.583,Z 1077.999,A -85,B 0,C 180,E1 5054.872,E2 5054.872} C_VEL
LIN {X 0,Y 665.827,Z 1064.493,A -85,B 0,C 180,E1 5057.161,E2 5057.161} C_VEL
LIN {X 0,Y 666.268,Z 1046.253,A -85,B 0,C 180,E1 5059.177,E2 5059.177} C_VEL
LIN {X 0,Y 666.663,Z 1022.883,A -85,B 0,C 180,E1 5060.917,E2 5060.917} C_VEL
LIN {X 0,Y 667.153,Z 996.582,A -85,B 0,C 180,E1 5062.201,E2 5062.201} C_VEL
LIN {X 0,Y 667.514,Z 968.131,A -85,B 0,C 180,E1 5063.006,E2 5063.006} C_VEL
LIN {X 0,Y 666.494,Z 932.193,A -85,B 0,C 180,E1 5063.488,E2 5063.488} C_VEL
LIN {X 0,Y 664.712,Z 923.03,A -85,B 0,C 180,E1 5063.674,E2 5063.674} C_VEL
LIN {X 0,Y 664.399,Z 923.03,A -85,B 0,C 180,E1 5068.532,E2 5068.532} C_VEL
LIN {X 0,Y 664.38,Z 923.03,A -85,B 0,C 180,E1 5073.086,E2 5073.086} C_VEL
LIN {X 0,Y 664.357,Z 923.03,A -85,B 0,C 180,E1 5077.89,E2 5077.89} C_VEL
LIN {X 0,Y 664.213,Z 923.03,A -85,B 0,C 180,E1 5083.269,E2 5083.269} C_VEL
LIN {X 0,Y 664.328,Z 923.03,A -85,B 0,C 180,E1 5088.717,E2 5088.717} C_VEL
LIN {X 0,Y 664.356,Z 923.03,A -85,B 0,C 180,E1 5093.735,E2 5093.735} C_VEL
LIN {X 0,Y 664.355,Z 923.03,A -85,B 0,C 180,E1 5098.447,E2 5098.447} C_VEL
LIN {X 0,Y 664.597,Z 923.03,A -85,B 0,C 180,E1 5102.942,E2 5102.942} C_VEL
LIN {X 0,Y 664.576,Z 923.03,A -85,B 0,C 180,E1 5107.25,E2 5107.25} C_VEL
LIN {X 0,Y 664.645,Z 923.03,A -85,B 0,C 180,E1 5112.799,E2 5112.799} C_VEL
LIN {X 0,Y 664.654,Z 923.03,A -85,B 0,C 180,E1 5118.182,E2 5118.182} C_VEL
LIN {X 0,Y 664.858,Z 923.03,A -85,B 0,C 180,E1 5123.464,E2 5123.464} C_VEL
LIN {X 0,Y 664.873,Z 923.03,A -85,B 0,C 180,E1 5128.686,E2 5128.686} C_VEL
LIN {X 0,Y 664.862,Z 923.03,A -85,B 0,C 180,E1 5132.594,E2 5132.594} C_VEL
LIN {X 0,Y 664.793,Z 923.03,A -85,B 0,C 180,E1 5136.514,E2 5136.514} C_VEL
LIN {X 0,Y 664.716,Z 923.03,A -85,B 0,C 180,E1 5141.793,E2 5141.793} C_VEL
LIN {X 0,Y 664.696,Z 923.03,A -85,B 0,C 180,E1 5147.285,E2 5147.285} C_VEL
LIN {X 0,Y 664.534,Z 923.03,A -85,B 0,C 180,E1 5152.726,E2 5152.726} C_VEL
LIN {X 0,Y 664.532,Z 923.03,A -85,B 0,C 180,E1 5157.519,E2 5157.519} C_VEL
LIN {X 0,Y 664.502,Z 923.03,A -85,B 0,C 180,E1 5163.06,E2 5163.06} C_VEL
LIN {X 0,Y 664.328,Z 923.03,A -85,B 0,C 180,E1 5167.871,E2 5167.871} C_VEL
LIN {X 0,Y 664.518,Z 923.03,A -85,B 0,C 180,E1 5173.306,E2 5173.306} C_VEL
LIN {X 0,Y 664.337,Z 923.03,A -85,B 0,C 180,E1 5178.726,E2 5178.726} C_VEL
LIN {X 0,Y 664.35,Z 923.03,A -85,B 0,C 180,E1 5183.743,E2 5183.743} C_VEL
LIN {X 0,Y 664.375,Z 923.03,A -85,B 0,C 180,E1 5188.456,E2 5188.456} C_VEL
LIN {X 0,Y 664.737,Z 923.661,A -85,B 0,C 180,E1 5193.849,E2 5193.849} C_VEL
LIN {X 0,Y 673.296,Z 950.529,A -85,B 0,C 180,E1 5194.669,E2 5194.669} C_VEL
LIN {X 0,Y 672.104,Z 990.527,A -85,B 0,C 180,E1 5195.83,E2 5195.83} C_VEL
LIN {X 0,Y 670.531,Z 1029.176,A -85,B 0,C 180,E1 5197.547,E2 5197.547} C_VEL
LIN {X 0,Y 668.929,Z 1063.538,A -85,B 0,C 180,E1 5199.662,E2 5199.662} C_VEL
LIN {X 0,Y 667.482,Z 1094.289,A -85,B 0,C 180,E1 5202.178,E2 5202.178} C_VEL
LIN {X 0,Y 666.477,Z 1119.924,A -85,B 0,C 180,E1 5204.935,E2 5204.935} C_VEL
LIN {X 0,Y 665.707,Z 1141.357,A -85,B 0,C 180,E1 5207.991,E2 5207.991} C_VEL
LIN {X 0,Y 665.308,Z 1157.599,A -85,B 0,C 180,E1 5211.198,E2 5211.198} C_VEL
LIN {X 0,Y 665.13,Z 1167.713,A -85,B 0,C 180,E1 5214.131,E2 5214.131} C_VEL
LIN {X 0,Y 665.046,Z 1173.969,A -85,B 0,C 180,E1 5217.394,E2 5217.394} C_VEL
LIN {X 0,Y 664.939,Z 1175.496,A -85,B 0,C 180,E1 5219.999,E2 5219.999} C_VEL
LIN {X 0,Y 665.096,Z 1173.853,A -85,B 0,C 180,E1 5222.603,E2 5222.603} C_VEL
LIN {X 0,Y 665.173,Z 1167.457,A -85,B 0,C 180,E1 5225.866,E2 5225.866} C_VEL
LIN {X 0,Y 665.303,Z 1155.796,A -85,B 0,C 180,E1 5229.147,E2 5229.147} C_VEL
LIN {X 0,Y 665.801,Z 1137.468,A -85,B 0,C 180,E1 5232.553,E2 5232.553} C_VEL
LIN {X 0,Y 666.679,Z 1114.129,A -85,B 0,C 180,E1 5235.67,E2 5235.67} C_VEL
LIN {X 0,Y 667.858,Z 1086.18,A -85,B 0,C 180,E1 5238.466,E2 5238.466} C_VEL
LIN {X 0,Y 669.295,Z 1055.505,A -85,B 0,C 180,E1 5240.8,E2 5240.8} C_VEL
LIN {X 0,Y 670.948,Z 1021.225,A -85,B 0,C 180,E1 5242.763,E2 5242.763} C_VEL
LIN {X 0,Y 671.676,Z 1001.807,A -85,B 0,C 180,E1 5243.642,E2 5243.642} C_VEL
LIN {X 0,Y 668.59,Z 986.576,A -85,B 0,C 180,E1 5244.345,E2 5244.345} C_VEL
LIN {X 0,Y 665.382,Z 970.982,A -85,B 0,C 180,E1 5244.964,E2 5244.964} C_VEL
LIN {X 0,Y 665.177,Z 948.91,A -85,B 0,C 180,E1 5245.544,E2 5245.544} C_VEL
LIN {X 0,Y 656.59,Z 923.03,A -85,B 0,C 180,E1 5246.378,E2 5246.378} C_VEL
LIN {X 0,Y 656.603,Z 923.03,A -85,B 0,C 180,E1 5251.958,E2 5251.958} C_VEL
LIN {X 0,Y 656.445,Z 923.03,A -85,B 0,C 180,E1 5256.761,E2 5256.761} C_VEL
LIN {X 0,Y 656.34,Z 923.03,A -85,B 0,C 180,E1 5262.569,E2 5262.569} C_VEL
LIN {X 0,Y 656.33,Z 923.03,A -85,B 0,C 180,E1 5268.132,E2 5268.132} C_VEL
LIN {X 0,Y 656.552,Z 923.03,A -85,B 0,C 180,E1 5273.661,E2 5273.661} C_VEL
LIN {X 0,Y 656.468,Z 923.03,A -85,B 0,C 180,E1 5278.393,E2 5278.393} C_VEL
LIN {X 0,Y 656.437,Z 923.145,A -85,B 0,C 180,E1 5282.971,E2 5282.971} C_VEL
LIN {X 0,Y 666.513,Z 953.544,A -85,B 0,C 180,E1 5283.661,E2 5283.661} C_VEL
LIN {X 0,Y 665.956,Z 1004.974,A -85,B 0,C 180,E1 5284.381,E2 5284.381} C_VEL
LIN {X 0,Y 664.915,Z 1044.08,A -85,B 0,C 180,E1 5285.424,E2 5285.424} C_VEL
LIN {X 0,Y 663.541,Z 1080.373,A -85,B 0,C 180,E1 5286.884,E2 5286.884} C_VEL
LIN {X 0,Y 661.913,Z 1114.793,A -85,B 0,C 180,E1 5288.863,E2 5288.863} C_VEL
LIN {X 0,Y 660.32,Z 1144.889,A -85,B 0,C 180,E1 5291.155,E2 5291.155} C_VEL
LIN {X 0,Y 659.011,Z 1172.165,A -85,B 0,C 180,E1 5293.871,E2 5293.871} C_VEL
LIN {X 0,Y 658.121,Z 1194.144,A -85,B 0,C 180,E1 5296.739,E2 5296.739} C_VEL
LIN {X 0,Y 657.504,Z 1212.976,A -85,B 0,C 180,E1 5300.087,E2 5300.087} C_VEL
LIN {X 0,Y 657.242,Z 1225.689,A -85,B 0,C 180,E1 5303.411,E2 5303.411} C_VEL
LIN {X 0,Y 657.176,Z 1231.97,A -85,B 0,C 180,E1 5306.057,E2 5306.057} C_VEL
LIN {X 0,Y 657.135,Z 1235.096,A -85,B 0,C 180,E1 5308.694,E2 5308.694} C_VEL
LIN {X 0,Y 657.271,Z 1235.079,A -85,B 0,C 180,E1 5311.329,E2 5311.329} C_VEL
LIN {X 0,Y 657.264,Z 1230.721,A -85,B 0,C 180,E1 5314.627,E2 5314.627} C_VEL
LIN {X 0,Y 657.373,Z 1221.231,A -85,B 0,C 180,E1 5317.939,E2 5317.939} C_VEL
LIN {X 0,Y 657.763,Z 1206.152,A -85,B 0,C 180,E1 5321.271,E2 5321.271} C_VEL
LIN {X 0,Y 658.485,Z 1184.41,A -85,B 0,C 180,E1 5324.632,E2 5324.632} C_VEL
LIN {X 0,Y 659.63,Z 1158.865,A -85,B 0,C 180,E1 5327.545,E2 5327.545} C_VEL
LIN {X 0,Y 661.092,Z 1129.938,A -85,B 0,C 180,E1 5330.062,E2 5330.062} C_VEL
LIN {X 0,Y 662.764,Z 1096.873,A -85,B 0,C 180,E1 5332.245,E2 5332.245} C_VEL
LIN {X 0,Y 664.348,Z 1061.375,A -85,B 0,C 180,E1 5333.956,E2 5333.956} C_VEL
LIN {X 0,Y 665.721,Z 1023.385,A -85,B 0,C 180,E1 5335.22,E2 5335.22} C_VEL
LIN {X 0,Y 666.57,Z 984.194,A -85,B 0,C 180,E1 5336.016,E2 5336.016} C_VEL
LIN {X 0,Y 666.048,Z 949.465,A -85,B 0,C 180,E1 5336.467,E2 5336.467} C_VEL
LIN {X 0,Y 656.472,Z 923.03,A -85,B 0,C 180,E1 5337.197,E2 5337.197} C_VEL
LIN {X 0,Y 656.556,Z 923.03,A -85,B 0,C 180,E1 5341.972,E2 5341.972} C_VEL
LIN {X 0,Y 656.488,Z 923.03,A -85,B 0,C 180,E1 5346.771,E2 5346.771} C_VEL
LIN {X 0,Y 656.355,Z 923.03,A -85,B 0,C 180,E1 5352.549,E2 5352.549} C_VEL
LIN {X 0,Y 656.348,Z 923.03,A -85,B 0,C 180,E1 5358.115,E2 5358.115} C_VEL
LIN {X 0,Y 656.543,Z 923.03,A -85,B 0,C 180,E1 5363.677,E2 5363.677} C_VEL
LIN {X 0,Y 656.48,Z 923.03,A -85,B 0,C 180,E1 5368.407,E2 5368.407} C_VEL
LIN {X 0,Y 656.577,Z 923.03,A -85,B 0,C 180,E1 5374.071,E2 5374.071} C_VEL
LIN {X 0,Y 656.621,Z 923.03,A -85,B 0,C 180,E1 5378.396,E2 5378.396} C_VEL
LIN {X 0,Y 656.521,Z 923.03,A -85,B 0,C 180,E1 5383.968,E2 5383.968} C_VEL
LIN {X 0,Y 656.864,Z 923.03,A -85,B 0,C 180,E1 5389.396,E2 5389.396} C_VEL
LIN {X 0,Y 656.814,Z 923.03,A -85,B 0,C 180,E1 5394.721,E2 5394.721} C_VEL
LIN {X 0,Y 656.805,Z 923.03,A -85,B 0,C 180,E1 5396.125,E2 5396.125} C_VEL
LIN {X 0,Y 659.75,Z 942.938,A -85,B 0,C 180,E1 5396.423,E2 5396.423} C_VEL
LIN {X 0,Y 659.753,Z 976.464,A -85,B 0,C 180,E1 5396.934,E2 5396.934} C_VEL
LIN {X 0,Y 659.37,Z 1004.942,A -85,B 0,C 180,E1 5397.867,E2 5397.867} C_VEL
LIN {X 0,Y 658.913,Z 1030.315,A -85,B 0,C 180,E1 5399.262,E2 5399.262} C_VEL
LIN {X 0,Y 658.435,Z 1053.016,A -85,B 0,C 180,E1 5401.152,E2 5401.152} C_VEL
LIN {X 0,Y 658.031,Z 1069.845,A -85,B 0,C 180,E1 5403.258,E2 5403.258} C_VEL
LIN {X 0,Y 657.682,Z 1081.811,A -85,B 0,C 180,E1 5405.605,E2 5405.605} C_VEL
LIN {X 0,Y 657.545,Z 1088.18,A -85,B 0,C 180,E1 5407.927,E2 5407.927} C_VEL
LIN {X 0,Y 657.476,Z 1089.686,A -85,B 0,C 180,E1 5410.596,E2 5410.596} C_VEL
LIN {X 0,Y 657.611,Z 1086.765,A -85,B 0,C 180,E1 5412.579,E2 5412.579} C_VEL
LIN {X 0,Y 657.764,Z 1078.839,A -85,B 0,C 180,E1 5414.931,E2 5414.931} C_VEL
LIN {X 0,Y 658.022,Z 1065.613,A -85,B 0,C 180,E1 5417.199,E2 5417.199} C_VEL
LIN {X 0,Y 658.504,Z 1046.924,A -85,B 0,C 180,E1 5419.288,E2 5419.288} C_VEL
LIN {X 0,Y 658.934,Z 1024.241,A -85,B 0,C 180,E1 5420.999,E2 5420.999} C_VEL
LIN {X 0,Y 659.469,Z 998.285,A -85,B 0,C 180,E1 5422.293,E2 5422.293} C_VEL
LIN {X 0,Y 659.792,Z 970.092,A -85,B 0,C 180,E1 5423.122,E2 5423.122} C_VEL
LIN {X 0,Y 658.927,Z 933.873,A -85,B 0,C 180,E1 5423.62,E2 5423.62} C_VEL
LIN {X 0,Y 656.796,Z 923.03,A -85,B 0,C 180,E1 5423.817,E2 5423.817} C_VEL
LIN {X 0,Y 656.443,Z 923.03,A -85,B 0,C 180,E1 5428.971,E2 5428.971} C_VEL
LIN {X 0,Y 656.411,Z 923.03,A -85,B 0,C 180,E1 5434.017,E2 5434.017} C_VEL
LIN {X 0,Y 656.416,Z 923.03,A -85,B 0,C 180,E1 5438.48,E2 5438.48} C_VEL
LIN {X 0,Y 656.305,Z 923.03,A -85,B 0,C 180,E1 5443.69,E2 5443.69} C_VEL
LIN {X 0,Y 656.364,Z 923.03,A -85,B 0,C 180,E1 5448.104,E2 5448.104} C_VEL
LIN {X 0,Y 656.465,Z 923.03,A -85,B 0,C 180,E1 5453.676,E2 5453.676} C_VEL
LIN {X 0,Y 656.458,Z 923.03,A -85,B 0,C 180,E1 5459.564,E2 5459.564} C_VEL
LIN {X 0,Y 656.686,Z 923.03,A -85,B 0,C 180,E1 5464.064,E2 5464.064} C_VEL
LIN {X 0,Y 656.68,Z 923.03,A -85,B 0,C 180,E1 5469.798,E2 5469.798} C_VEL
LIN {X 0,Y 656.685,Z 923.03,A -85,B 0,C 180,E1 5475.124,E2 5475.124} C_VEL
LIN {X 0,Y 656.869,Z 923.03,A -85,B 0,C 180,E1 5480.722,E2 5480.722} C_VEL
LIN {X 0,Y 657.026,Z 923.03,A -85,B 0,C 180,E1 5486.032,E2 5486.032} C_VEL
LIN {X 0,Y 657.161,Z 923.03,A -85,B 0,C 180,E1 5491.306,E2 5491.306} C_VEL
LIN {X 0,Y 656.885,Z 923.03,A -85,B 0,C 180,E1 5496.592,E2 5496.592} C_VEL
LIN {X 0,Y 656.808,Z 923.03,A -85,B 0,C 180,E1 5501.937,E2 5501.937} C_VEL
LIN {X 0,Y 656.798,Z 923.03,A -85,B 0,C 180,E1 5507.389,E2 5507.389} C_VEL
LIN {X 0,Y 656.625,Z 923.03,A -85,B 0,C 180,E1 5513.016,E2 5513.016} C_VEL
LIN {X 0,Y 656.628,Z 923.03,A -85,B 0,C 180,E1 5517.388,E2 5517.388} C_VEL
LIN {X 0,Y 656.591,Z 923.03,A -85,B 0,C 180,E1 5521.943,E2 5521.943} C_VEL
LIN {X 0,Y 656.469,Z 923.03,A -85,B 0,C 180,E1 5526.743,E2 5526.743} C_VEL
LIN {X 0,Y 656.543,Z 923.03,A -85,B 0,C 180,E1 5532.563,E2 5532.563} C_VEL
LIN {X 0,Y 656.414,Z 923.03,A -85,B 0,C 180,E1 5537.424,E2 5537.424} C_VEL
LIN {X 0,Y 656.451,Z 923.03,A -85,B 0,C 180,E1 5543.236,E2 5543.236} C_VEL
LIN {X 0,Y 656.487,Z 923.03,A -85,B 0,C 180,E1 5548.362,E2 5548.362} C_VEL
LIN {X 0,Y 656.78,Z 923.03,A -85,B 0,C 180,E1 5553.523,E2 5553.523} C_VEL
LIN {X 0,Y 666.011,Z 953.26,A -85,B 0,C 180,E1 5554.462,E2 5554.462} C_VEL
LIN {X 0,Y 664.641,Z 993.922,A -85,B 0,C 180,E1 5555.693,E2 5555.693} C_VEL
LIN {X 0,Y 663.074,Z 1030.493,A -85,B 0,C 180,E1 5557.356,E2 5557.356} C_VEL
LIN {X 0,Y 661.341,Z 1064.292,A -85,B 0,C 180,E1 5559.475,E2 5559.475} C_VEL
LIN {X 0,Y 659.815,Z 1094.648,A -85,B 0,C 180,E1 5562,E2 5562} C_VEL
LIN {X 0,Y 658.695,Z 1120.763,A -85,B 0,C 180,E1 5564.859,E2 5564.859} C_VEL
LIN {X 0,Y 657.857,Z 1142.662,A -85,B 0,C 180,E1 5568.068,E2 5568.068} C_VEL
LIN {X 0,Y 657.424,Z 1157.788,A -85,B 0,C 180,E1 5571.139,E2 5571.139} C_VEL
LIN {X 0,Y 657.248,Z 1167.712,A -85,B 0,C 180,E1 5574.06,E2 5574.06} C_VEL
LIN {X 0,Y 657.143,Z 1173.969,A -85,B 0,C 180,E1 5577.363,E2 5577.363} C_VEL
LIN {X 0,Y 657.06,Z 1175.496,A -85,B 0,C 180,E1 5579.999,E2 5579.999} C_VEL
LIN {X 0,Y 657.192,Z 1173.855,A -85,B 0,C 180,E1 5582.634,E2 5582.634} C_VEL
LIN {X 0,Y 657.298,Z 1167.46,A -85,B 0,C 180,E1 5585.937,E2 5585.937} C_VEL
LIN {X 0,Y 657.433,Z 1155.798,A -85,B 0,C 180,E1 5589.257,E2 5589.257} C_VEL
LIN {X 0,Y 657.997,Z 1137.474,A -85,B 0,C 180,E1 5592.704,E2 5592.704} C_VEL
LIN {X 0,Y 658.9,Z 1115.141,A -85,B 0,C 180,E1 5595.743,E2 5595.743} C_VEL
LIN {X 0,Y 660.143,Z 1088.089,A -85,B 0,C 180,E1 5598.521,E2 5598.521} C_VEL
LIN {X 0,Y 661.727,Z 1057.593,A -85,B 0,C 180,E1 5600.907,E2 5600.907} C_VEL
LIN {X 0,Y 663.518,Z 1022.723,A -85,B 0,C 180,E1 5602.953,E2 5602.953} C_VEL
LIN {X 0,Y 664.918,Z 987.168,A -85,B 0,C 180,E1 5604.445,E2 5604.445} C_VEL
LIN {X 0,Y 665.382,Z 970.982,A -85,B 0,C 180,E1 5604.964,E2 5604.964} C_VEL
LIN {X 0,Y 662.607,Z 960.563,A -85,B 0,C 180,E1 5605.354,E2 5605.354} C_VEL
LIN {X 0,Y 657.687,Z 950.56,A -85,B 0,C 180,E1 5605.764,E2 5605.764} C_VEL
LIN {X 0,Y 648.671,Z 923.03,A -85,B 0,C 180,E1 5606.642,E2 5606.642} C_VEL
LIN {X 0,Y 648.629,Z 923.03,A -85,B 0,C 180,E1 5612.398,E2 5612.398} C_VEL
LIN {X 0,Y 648.44,Z 923.03,A -85,B 0,C 180,E1 5617.623,E2 5617.623} C_VEL
LIN {X 0,Y 648.436,Z 923.03,A -85,B 0,C 180,E1 5622.515,E2 5622.515} C_VEL
LIN {X 0,Y 648.42,Z 923.03,A -85,B 0,C 180,E1 5628.22,E2 5628.22} C_VEL
LIN {X 0,Y 648.529,Z 923.03,A -85,B 0,C 180,E1 5632.732,E2 5632.732} C_VEL
LIN {X 0,Y 648.531,Z 923.03,A -85,B 0,C 180,E1 5637.612,E2 5637.612} C_VEL
LIN {X 0,Y 648.596,Z 923.83,A -85,B 0,C 180,E1 5642.702,E2 5642.702} C_VEL
LIN {X 0,Y 659.155,Z 955.172,A -85,B 0,C 180,E1 5643.436,E2 5643.436} C_VEL
LIN {X 0,Y 658.603,Z 1003.498,A -85,B 0,C 180,E1 5644.121,E2 5644.121} C_VEL
LIN {X 0,Y 657.423,Z 1043.612,A -85,B 0,C 180,E1 5645.195,E2 5645.195} C_VEL
LIN {X 0,Y 655.949,Z 1080.416,A -85,B 0,C 180,E1 5646.69,E2 5646.69} C_VEL
LIN {X 0,Y 654.348,Z 1115.775,A -85,B 0,C 180,E1 5648.687,E2 5648.687} C_VEL
LIN {X 0,Y 652.711,Z 1144.888,A -85,B 0,C 180,E1 5650.927,E2 5650.927} C_VEL
LIN {X 0,Y 651.318,Z 1172.163,A -85,B 0,C 180,E1 5653.676,E2 5653.676} C_VEL
LIN {X 0,Y 650.327,Z 1194.144,A -85,B 0,C 180,E1 5656.577,E2 5656.577} C_VEL
LIN {X 0,Y 649.65,Z 1212.976,A -85,B 0,C 180,E1 5659.966,E2 5659.966} C_VEL
LIN {X 0,Y 649.379,Z 1225.689,A -85,B 0,C 180,E1 5663.331,E2 5663.331} C_VEL
LIN {X 0,Y 649.279,Z 1231.969,A -85,B 0,C 180,E1 5666.008,E2 5666.008} C_VEL
LIN {X 0,Y 649.246,Z 1235.096,A -85,B 0,C 180,E1 5668.678,E2 5668.678} C_VEL
LIN {X 0,Y 649.369,Z 1235.08,A -85,B 0,C 180,E1 5671.345,E2 5671.345} C_VEL
LIN {X 0,Y 649.364,Z 1230.721,A -85,B 0,C 180,E1 5674.683,E2 5674.683} C_VEL
LIN {X 0,Y 649.519,Z 1221.231,A -85,B 0,C 180,E1 5678.035,E2 5678.035} C_VEL
LIN {X 0,Y 649.914,Z 1206.152,A -85,B 0,C 180,E1 5681.409,E2 5681.409} C_VEL
LIN {X 0,Y 650.713,Z 1184.408,A -85,B 0,C 180,E1 5684.811,E2 5684.811} C_VEL
LIN {X 0,Y 651.918,Z 1159.331,A -85,B 0,C 180,E1 5687.713,E2 5687.713} C_VEL
LIN {X 0,Y 653.521,Z 1129.935,A -85,B 0,C 180,E1 5690.304,E2 5690.304} C_VEL
LIN {X 0,Y 655.25,Z 1096.468,A -85,B 0,C 180,E1 5692.498,E2 5692.498} C_VEL
LIN {X 0,Y 656.957,Z 1059.068,A -85,B 0,C 180,E1 5694.287,E2 5694.287} C_VEL
LIN {X 0,Y 658.455,Z 1019.911,A -85,B 0,C 180,E1 5695.568,E2 5695.568} C_VEL
LIN {X 0,Y 659.321,Z 980.332,A -85,B 0,C 180,E1 5696.34,E2 5696.34} C_VEL
LIN {X 0,Y 658.863,Z 951.483,A -85,B 0,C 180,E1 5696.724,E2 5696.724} C_VEL
LIN {X 0,Y 648.566,Z 923.03,A -85,B 0,C 180,E1 5697.514,E2 5697.514} C_VEL
LIN {X 0,Y 648.601,Z 923.03,A -85,B 0,C 180,E1 5702.412,E2 5702.412} C_VEL
LIN {X 0,Y 648.485,Z 923.03,A -85,B 0,C 180,E1 5707.605,E2 5707.605} C_VEL
LIN {X 0,Y 648.454,Z 923.03,A -85,B 0,C 180,E1 5712.526,E2 5712.526} C_VEL
LIN {X 0,Y 648.434,Z 923.03,A -85,B 0,C 180,E1 5718.233,E2 5718.233} C_VEL
LIN {X 0,Y 648.51,Z 923.03,A -85,B 0,C 180,E1 5722.713,E2 5722.713} C_VEL
LIN {X 0,Y 648.516,Z 923.03,A -85,B 0,C 180,E1 5727.595,E2 5727.595} C_VEL
LIN {X 0,Y 648.612,Z 923.03,A -85,B 0,C 180,E1 5732.304,E2 5732.304} C_VEL
LIN {X 0,Y 648.723,Z 923.03,A -85,B 0,C 180,E1 5736.674,E2 5736.674} C_VEL
LIN {X 0,Y 648.604,Z 923.03,A -85,B 0,C 180,E1 5740.965,E2 5740.965} C_VEL
LIN {X 0,Y 648.733,Z 923.03,A -85,B 0,C 180,E1 5746.532,E2 5746.532} C_VEL
LIN {X 0,Y 648.968,Z 923.03,A -85,B 0,C 180,E1 5750.621,E2 5750.621} C_VEL
LIN {X 0,Y 648.869,Z 923.03,A -85,B 0,C 180,E1 5755.953,E2 5755.953} C_VEL
LIN {X 0,Y 652.097,Z 944.96,A -85,B 0,C 180,E1 5756.292,E2 5756.292} C_VEL
LIN {X 0,Y 652.057,Z 978.425,A -85,B 0,C 180,E1 5756.821,E2 5756.821} C_VEL
LIN {X 0,Y 651.625,Z 1008.151,A -85,B 0,C 180,E1 5757.842,E2 5757.842} C_VEL
LIN {X 0,Y 651.138,Z 1034,A -85,B 0,C 180,E1 5759.337,E2 5759.337} C_VEL
LIN {X 0,Y 650.642,Z 1054.991,A -85,B 0,C 180,E1 5761.166,E2 5761.166} C_VEL
LIN {X 0,Y 650.235,Z 1071.703,A -85,B 0,C 180,E1 5763.332,E2 5763.332} C_VEL
LIN {X 0,Y 649.848,Z 1083.196,A -85,B 0,C 180,E1 5765.673,E2 5765.673} C_VEL
LIN {X 0,Y 649.72,Z 1089.318,A -85,B 0,C 180,E1 5768.023,E2 5768.023} C_VEL
LIN {X 0,Y 649.669,Z 1090.694,A -85,B 0,C 180,E1 5769.372,E2 5769.372} C_VEL
LIN {X 0,Y 649.748,Z 1088.783,A -85,B 0,C 180,E1 5772.083,E2 5772.083} C_VEL
LIN {X 0,Y 649.884,Z 1081.877,A -85,B 0,C 180,E1 5774.476,E2 5774.476} C_VEL
LIN {X 0,Y 650.221,Z 1069.163,A -85,B 0,C 180,E1 5776.889,E2 5776.889} C_VEL
LIN {X 0,Y 650.603,Z 1050.751,A -85,B 0,C 180,E1 5779.101,E2 5779.101} C_VEL
LIN {X 0,Y 651.192,Z 1028.389,A -85,B 0,C 180,E1 5780.904,E2 5780.904} C_VEL
LIN {X 0,Y 651.744,Z 1002.013,A -85,B 0,C 180,E1 5782.302,E2 5782.302} C_VEL
LIN {X 0,Y 652.141,Z 972.346,A -85,B 0,C 180,E1 5783.232,E2 5783.232} C_VEL
LIN {X 0,Y 651.14,Z 934.241,A -85,B 0,C 180,E1 5783.773,E2 5783.773} C_VEL
LIN {X 0,Y 648.881,Z 923.03,A -85,B 0,C 180,E1 5783.974,E2 5783.974} C_VEL
LIN {X 0,Y 648.524,Z 923.03,A -85,B 0,C 180,E1 5789.297,E2 5789.297} C_VEL
LIN {X 0,Y 648.54,Z 923.03,A -85,B 0,C 180,E1 5794.002,E2 5794.002} C_VEL
LIN {X 0,Y 648.439,Z 923.03,A -85,B 0,C 180,E1 5799.722,E2 5799.722} C_VEL
LIN {X 0,Y 648.408,Z 923.03,A -85,B 0,C 180,E1 5804.36,E2 5804.36} C_VEL
LIN {X 0,Y 648.5,Z 923.03,A -85,B 0,C 180,E1 5809.263,E2 5809.263} C_VEL
LIN {X 0,Y 648.52,Z 923.03,A -85,B 0,C 180,E1 5814.642,E2 5814.642} C_VEL
LIN {X 0,Y 648.581,Z 923.03,A -85,B 0,C 180,E1 5819.55,E2 5819.55} C_VEL
LIN {X 0,Y 648.767,Z 923.03,A -85,B 0,C 180,E1 5823.723,E2 5823.723} C_VEL
LIN {X 0,Y 648.706,Z 923.03,A -85,B 0,C 180,E1 5828.715,E2 5828.715} C_VEL
LIN {X 0,Y 648.813,Z 923.03,A -85,B 0,C 180,E1 5833.76,E2 5833.76} C_VEL
LIN {X 0,Y 648.919,Z 923.03,A -85,B 0,C 180,E1 5839.253,E2 5839.253} C_VEL
LIN {X 0,Y 649.006,Z 923.03,A -85,B 0,C 180,E1 5844.645,E2 5844.645} C_VEL
LIN {X 0,Y 649.076,Z 923.03,A -85,B 0,C 180,E1 5848.654,E2 5848.654} C_VEL
LIN {X 0,Y 649.064,Z 923.03,A -85,B 0,C 180,E1 5852.657,E2 5852.657} C_VEL
LIN {X 0,Y 648.996,Z 923.03,A -85,B 0,C 180,E1 5856.673,E2 5856.673} C_VEL
LIN {X 0,Y 648.898,Z 923.03,A -85,B 0,C 180,E1 5862.085,E2 5862.085} C_VEL
LIN {X 0,Y 648.862,Z 923.03,A -85,B 0,C 180,E1 5867.609,E2 5867.609} C_VEL
LIN {X 0,Y 648.696,Z 923.03,A -85,B 0,C 180,E1 5873.314,E2 5873.314} C_VEL
LIN {X 0,Y 648.678,Z 923.03,A -85,B 0,C 180,E1 5877.752,E2 5877.752} C_VEL
LIN {X 0,Y 648.608,Z 923.03,A -85,B 0,C 180,E1 5882.993,E2 5882.993} C_VEL
LIN {X 0,Y 648.471,Z 923.03,A -85,B 0,C 180,E1 5887.598,E2 5887.598} C_VEL
LIN {X 0,Y 648.633,Z 923.03,A -85,B 0,C 180,E1 5892.48,E2 5892.48} C_VEL
LIN {X 0,Y 648.509,Z 923.03,A -85,B 0,C 180,E1 5897.487,E2 5897.487} C_VEL
LIN {X 0,Y 648.482,Z 923.03,A -85,B 0,C 180,E1 5902.708,E2 5902.708} C_VEL
LIN {X 0,Y 648.498,Z 923.03,A -85,B 0,C 180,E1 5907.591,E2 5907.591} C_VEL
LIN {X 0,Y 648.827,Z 923.03,A -85,B 0,C 180,E1 5913.193,E2 5913.193} C_VEL
LIN {X 0,Y 658.73,Z 953.812,A -85,B 0,C 180,E1 5914.201,E2 5914.201} C_VEL
LIN {X 0,Y 657.267,Z 994.545,A -85,B 0,C 180,E1 5915.453,E2 5915.453} C_VEL
LIN {X 0,Y 655.578,Z 1031.824,A -85,B 0,C 180,E1 5917.176,E2 5917.176} C_VEL
LIN {X 0,Y 653.813,Z 1064.272,A -85,B 0,C 180,E1 5919.228,E2 5919.228} C_VEL
LIN {X 0,Y 652.222,Z 1094.14,A -85,B 0,C 180,E1 5921.734,E2 5921.734} C_VEL
LIN {X 0,Y 651.031,Z 1119.478,A -85,B 0,C 180,E1 5924.514,E2 5924.514} C_VEL
LIN {X 0,Y 650.04,Z 1140.538,A -85,B 0,C 180,E1 5927.559,E2 5927.559} C_VEL
LIN {X 0,Y 649.58,Z 1156.154,A -85,B 0,C 180,E1 5930.627,E2 5930.627} C_VEL
LIN {X 0,Y 649.364,Z 1167.711,A -85,B 0,C 180,E1 5933.988,E2 5933.988} C_VEL
LIN {X 0,Y 649.255,Z 1173.969,A -85,B 0,C 180,E1 5937.331,E2 5937.331} C_VEL
LIN {X 0,Y 649.161,Z 1175.496,A -85,B 0,C 180,E1 5939.999,E2 5939.999} C_VEL
LIN {X 0,Y 649.312,Z 1173.856,A -85,B 0,C 180,E1 5942.666,E2 5942.666} C_VEL
LIN {X 0,Y 649.419,Z 1167.463,A -85,B 0,C 180,E1 5946.009,E2 5946.009} C_VEL
LIN {X 0,Y 649.563,Z 1155.8,A -85,B 0,C 180,E1 5949.37,E2 5949.37} C_VEL
LIN {X 0,Y 650.135,Z 1138.512,A -85,B 0,C 180,E1 5952.697,E2 5952.697} C_VEL
LIN {X 0,Y 651.177,Z 1114.597,A -85,B 0,C 180,E1 5955.999,E2 5955.999} C_VEL
LIN {X 0,Y 652.58,Z 1087.309,A -85,B 0,C 180,E1 5958.814,E2 5958.814} C_VEL
LIN {X 0,Y 654.269,Z 1056.361,A -85,B 0,C 180,E1 5961.236,E2 5961.236} C_VEL
LIN {X 0,Y 656.037,Z 1022.032,A -85,B 0,C 180,E1 5963.23,E2 5963.23} C_VEL
LIN {X 0,Y 657.551,Z 985.916,A -85,B 0,C 180,E1 5964.738,E2 5964.738} C_VEL
LIN {X 0,Y 657.837,Z 950.96,A -85,B 0,C 180,E1 5965.75,E2 5965.75} C_VEL
LIN {X 0,Y 657.687,Z 950.56,A -85,B 0,C 180,E1 5965.764,E2 5965.764} C_VEL
LIN {X 0,Y 650.611,Z 942.287,A -85,B 0,C 180,E1 5966.195,E2 5966.195} C_VEL
LIN {X 0,Y 644.355,Z 935.069,A -85,B 0,C 180,E1 5966.552,E2 5966.552} C_VEL
LIN {X 0,Y 643.88,Z 933.758,A -85,B 0,C 180,E1 5966.593,E2 5966.593} C_VEL
LIN {X 0,Y 640.753,Z 923.03,A -85,B 0,C 180,E1 5966.942,E2 5966.942} C_VEL
LIN {X 0,Y 640.708,Z 923.03,A -85,B 0,C 180,E1 5971.922,E2 5971.922} C_VEL
LIN {X 0,Y 640.536,Z 923.03,A -85,B 0,C 180,E1 5976.696,E2 5976.696} C_VEL
LIN {X 0,Y 640.512,Z 923.03,A -85,B 0,C 180,E1 5981.342,E2 5981.342} C_VEL
LIN {X 0,Y 640.52,Z 923.03,A -85,B 0,C 180,E1 5986.997,E2 5986.997} C_VEL
LIN {X 0,Y 640.578,Z 923.03,A -85,B 0,C 180,E1 5992.189,E2 5992.189} C_VEL
LIN {X 0,Y 640.642,Z 923.03,A -85,B 0,C 180,E1 5997.163,E2 5997.163} C_VEL
LIN {X 0,Y 640.652,Z 923.03,A -85,B 0,C 180,E1 6002.388,E2 6002.388} C_VEL
LIN {X 0,Y 651.788,Z 956.738,A -85,B 0,C 180,E1 6003.205,E2 6003.205} C_VEL
LIN {X 0,Y 651.144,Z 1004.07,A -85,B 0,C 180,E1 6003.897,E2 6003.897} C_VEL
LIN {X 0,Y 649.91,Z 1043.718,A -85,B 0,C 180,E1 6004.982,E2 6004.982} C_VEL
LIN {X 0,Y 648.367,Z 1080.385,A -85,B 0,C 180,E1 6006.492,E2 6006.492} C_VEL
LIN {X 0,Y 646.656,Z 1115.578,A -85,B 0,C 180,E1 6008.502,E2 6008.502} C_VEL
LIN {X 0,Y 644.983,Z 1146.635,A -85,B 0,C 180,E1 6010.867,E2 6010.867} C_VEL
LIN {X 0,Y 643.588,Z 1172.162,A -85,B 0,C 180,E1 6013.474,E2 6013.474} C_VEL
LIN {X 0,Y 642.437,Z 1195.599,A -85,B 0,C 180,E1 6016.642,E2 6016.642} C_VEL
LIN {X 0,Y 641.795,Z 1212.975,A -85,B 0,C 180,E1 6019.842,E2 6019.842} C_VEL
LIN {X 0,Y 641.485,Z 1225.688,A -85,B 0,C 180,E1 6023.249,E2 6023.249} C_VEL
LIN {X 0,Y 641.383,Z 1231.968,A -85,B 0,C 180,E1 6025.959,E2 6025.959} C_VEL
LIN {X 0,Y 641.345,Z 1235.097,A -85,B 0,C 180,E1 6028.662,E2 6028.662} C_VEL
LIN {X 0,Y 641.466,Z 1235.08,A -85,B 0,C 180,E1 6031.362,E2 6031.362} C_VEL
LIN {X 0,Y 641.48,Z 1230.72,A -85,B 0,C 180,E1 6034.741,E2 6034.741} C_VEL
LIN {X 0,Y 641.64,Z 1221.231,A -85,B 0,C 180,E1 6038.135,E2 6038.135} C_VEL
LIN {X 0,Y 642.067,Z 1206.153,A -85,B 0,C 180,E1 6041.551,E2 6041.551} C_VEL
LIN {X 0,Y 642.966,Z 1184.407,A -85,B 0,C 180,E1 6044.993,E2 6044.993} C_VEL
LIN {X 0,Y 644.306,Z 1158.338,A -85,B 0,C 180,E1 6048.03,E2 6048.03} C_VEL
LIN {X 0,Y 645.926,Z 1129.308,A -85,B 0,C 180,E1 6050.554,E2 6050.554} C_VEL
LIN {X 0,Y 647.754,Z 1095.104,A -85,B 0,C 180,E1 6052.795,E2 6052.795} C_VEL
LIN {X 0,Y 649.558,Z 1057.858,A -85,B 0,C 180,E1 6054.582,E2 6054.582} C_VEL
LIN {X 0,Y 651.144,Z 1019.879,A -85,B 0,C 180,E1 6055.833,E2 6055.833} C_VEL
LIN {X 0,Y 652.096,Z 981.232,A -85,B 0,C 180,E1 6056.604,E2 6056.604} C_VEL
LIN {X 0,Y 651.798,Z 953.756,A -85,B 0,C 180,E1 6056.972,E2 6056.972} C_VEL
LIN {X 0,Y 640.651,Z 923.03,A -85,B 0,C 180,E1 6057.87,E2 6057.87} C_VEL
LIN {X 0,Y 640.706,Z 923.03,A -85,B 0,C 180,E1 6062.861,E2 6062.861} C_VEL
LIN {X 0,Y 640.559,Z 923.03,A -85,B 0,C 180,E1 6067.843,E2 6067.843} C_VEL
LIN {X 0,Y 640.543,Z 923.03,A -85,B 0,C 180,E1 6073.179,E2 6073.179} C_VEL
LIN {X 0,Y 640.509,Z 923.03,A -85,B 0,C 180,E1 6078.658,E2 6078.658} C_VEL
LIN {X 0,Y 640.615,Z 923.03,A -85,B 0,C 180,E1 6083.866,E2 6083.866} C_VEL
LIN {X 0,Y 640.598,Z 923.03,A -85,B 0,C 180,E1 6088.74,E2 6088.74} C_VEL
LIN {X 0,Y 640.755,Z 923.03,A -85,B 0,C 180,E1 6093.673,E2 6093.673} C_VEL
LIN {X 0,Y 640.773,Z 923.03,A -85,B 0,C 180,E1 6097.834,E2 6097.834} C_VEL
LIN {X 0,Y 640.67,Z 923.03,A -85,B 0,C 180,E1 6103.56,E2 6103.56} C_VEL
LIN {X 0,Y 641.031,Z 923.03,A -85,B 0,C 180,E1 6109.131,E2 6109.131} C_VEL
LIN {X 0,Y 641.009,Z 923.03,A -85,B 0,C 180,E1 6114.591,E2 6114.591} C_VEL
LIN {X 0,Y 640.992,Z 923.03,A -85,B 0,C 180,E1 6115.777,E2 6115.777} C_VEL
LIN {X 0,Y 644.401,Z 944.288,A -85,B 0,C 180,E1 6116.123,E2 6116.123} C_VEL
LIN {X 0,Y 644.394,Z 978.268,A -85,B 0,C 180,E1 6116.65,E2 6116.65} C_VEL
LIN {X 0,Y 643.958,Z 1007.767,A -85,B 0,C 180,E1 6117.648,E2 6117.648} C_VEL
LIN {X 0,Y 643.445,Z 1032.894,A -85,B 0,C 180,E1 6119.076,E2 6119.076} C_VEL
LIN {X 0,Y 642.977,Z 1053.765,A -85,B 0,C 180,E1 6120.843,E2 6120.843} C_VEL
LIN {X 0,Y 642.47,Z 1071.284,A -85,B 0,C 180,E1 6123.035,E2 6123.035} C_VEL
LIN {X 0,Y 642.07,Z 1083.307,A -85,B 0,C 180,E1 6125.403,E2 6125.403} C_VEL
LIN {X 0,Y 641.926,Z 1089.266,A -85,B 0,C 180,E1 6127.44,E2 6127.44} C_VEL
LIN {X 0,Y 641.831,Z 1091.653,A -85,B 0,C 180,E1 6129.487,E2 6129.487} C_VEL
LIN {X 0,Y 641.906,Z 1089.461,A -85,B 0,C 180,E1 6132.233,E2 6132.233} C_VEL
LIN {X 0,Y 642.088,Z 1082.242,A -85,B 0,C 180,E1 6134.656,E2 6134.656} C_VEL
LIN {X 0,Y 642.438,Z 1069.103,A -85,B 0,C 180,E1 6137.094,E2 6137.094} C_VEL
LIN {X 0,Y 642.85,Z 1051.395,A -85,B 0,C 180,E1 6139.215,E2 6139.215} C_VEL
LIN {X 0,Y 643.417,Z 1028.302,A -85,B 0,C 180,E1 6141.078,E2 6141.078} C_VEL
LIN {X 0,Y 644.043,Z 1001.069,A -85,B 0,C 180,E1 6142.505,E2 6142.505} C_VEL
LIN {X 0,Y 644.454,Z 972.402,A -85,B 0,C 180,E1 6143.387,E2 6143.387} C_VEL
LIN {X 0,Y 643.646,Z 936.299,A -85,B 0,C 180,E1 6143.904,E2 6143.904} C_VEL
LIN {X 0,Y 640.958,Z 923.03,A -85,B 0,C 180,E1 6144.187,E2 6144.187} C_VEL
LIN {X 0,Y 640.609,Z 923.03,A -85,B 0,C 180,E1 6149.695,E2 6149.695} C_VEL
LIN {X 0,Y 640.6,Z 923.03,A -85,B 0,C 180,E1 6154.483,E2 6154.483} C_VEL
LIN {X 0,Y 640.537,Z 923.03,A -85,B 0,C 180,E1 6159.567,E2 6159.567} C_VEL
LIN {X 0,Y 640.497,Z 923.03,A -85,B 0,C 180,E1 6165.056,E2 6165.056} C_VEL
LIN {X 0,Y 640.586,Z 923.03,A -85,B 0,C 180,E1 6170.427,E2 6170.427} C_VEL
LIN {X 0,Y 640.583,Z 923.03,A -85,B 0,C 180,E1 6175.655,E2 6175.655} C_VEL
LIN {X 0,Y 640.719,Z 923.03,A -85,B 0,C 180,E1 6180.768,E2 6180.768} C_VEL
LIN {X 0,Y 640.831,Z 923.03,A -85,B 0,C 180,E1 6184.874,E2 6184.874} C_VEL
LIN {X 0,Y 640.843,Z 923.03,A -85,B 0,C 180,E1 6190.713,E2 6190.713} C_VEL
LIN {X 0,Y 640.909,Z 923.03,A -85,B 0,C 180,E1 6195.172,E2 6195.172} C_VEL
LIN {X 0,Y 641.042,Z 923.03,A -85,B 0,C 180,E1 6200.491,E2 6200.491} C_VEL
LIN {X 0,Y 641.227,Z 923.03,A -85,B 0,C 180,E1 6205.934,E2 6205.934} C_VEL
LIN {X 0,Y 641.364,Z 923.03,A -85,B 0,C 180,E1 6211.338,E2 6211.338} C_VEL
LIN {X 0,Y 641.087,Z 923.03,A -85,B 0,C 180,E1 6216.756,E2 6216.756} C_VEL
LIN {X 0,Y 640.979,Z 923.03,A -85,B 0,C 180,E1 6222.236,E2 6222.236} C_VEL
LIN {X 0,Y 640.928,Z 923.03,A -85,B 0,C 180,E1 6227.834,E2 6227.834} C_VEL
LIN {X 0,Y 640.807,Z 923.03,A -85,B 0,C 180,E1 6233.119,E2 6233.119} C_VEL
LIN {X 0,Y 640.73,Z 923.03,A -85,B 0,C 180,E1 6238.127,E2 6238.127} C_VEL
LIN {X 0,Y 640.735,Z 923.03,A -85,B 0,C 180,E1 6242.831,E2 6242.831} C_VEL
LIN {X 0,Y 640.549,Z 923.03,A -85,B 0,C 180,E1 6247.813,E2 6247.813} C_VEL
LIN {X 0,Y 640.74,Z 923.03,A -85,B 0,C 180,E1 6253.13,E2 6253.13} C_VEL
LIN {X 0,Y 640.587,Z 923.03,A -85,B 0,C 180,E1 6258.988,E2 6258.988} C_VEL
LIN {X 0,Y 640.542,Z 923.03,A -85,B 0,C 180,E1 6263.857,E2 6263.857} C_VEL
LIN {X 0,Y 640.591,Z 923.03,A -85,B 0,C 180,E1 6268.736,E2 6268.736} C_VEL
LIN {X 0,Y 640.879,Z 923.03,A -85,B 0,C 180,E1 6272.874,E2 6272.874} C_VEL
LIN {X 0,Y 651.426,Z 956.244,A -85,B 0,C 180,E1 6273.98,E2 6273.98} C_VEL
LIN {X 0,Y 649.891,Z 996.381,A -85,B 0,C 180,E1 6275.257,E2 6275.257} C_VEL
LIN {X 0,Y 648.1,Z 1032.856,A -85,B 0,C 180,E1 6276.977,E2 6276.977} C_VEL
LIN {X 0,Y 646.157,Z 1066.708,A -85,B 0,C 180,E1 6279.168,E2 6279.168} C_VEL
LIN {X 0,Y 644.416,Z 1097.096,A -85,B 0,C 180,E1 6281.797,E2 6281.797} C_VEL
LIN {X 0,Y 643.069,Z 1123.54,A -85,B 0,C 180,E1 6284.843,E2 6284.843} C_VEL
LIN {X 0,Y 642.137,Z 1144.619,A -85,B 0,C 180,E1 6288.116,E2 6288.116} C_VEL
LIN {X 0,Y 641.681,Z 1159.695,A -85,B 0,C 180,E1 6291.401,E2 6291.401} C_VEL
LIN {X 0,Y 641.462,Z 1169.31,A -85,B 0,C 180,E1 6294.592,E2 6294.592} C_VEL
LIN {X 0,Y 641.352,Z 1173.97,A -85,B 0,C 180,E1 6297.298,E2 6297.298} C_VEL
LIN {X 0,Y 641.261,Z 1175.496,A -85,B 0,C 180,E1 6299.999,E2 6299.999} C_VEL
LIN {X 0,Y 641.409,Z 1173.855,A -85,B 0,C 180,E1 6302.699,E2 6302.699} C_VEL
LIN {X 0,Y 641.521,Z 1167.466,A -85,B 0,C 180,E1 6306.083,E2 6306.083} C_VEL
LIN {X 0,Y 641.703,Z 1155.801,A -85,B 0,C 180,E1 6309.486,E2 6309.486} C_VEL
LIN {X 0,Y 642.355,Z 1137.883,A -85,B 0,C 180,E1 6312.956,E2 6312.956} C_VEL
LIN {X 0,Y 643.442,Z 1114.973,A -85,B 0,C 180,E1 6316.152,E2 6316.152} C_VEL
LIN {X 0,Y 644.939,Z 1088.032,A -85,B 0,C 180,E1 6318.977,E2 6318.977} C_VEL
LIN {X 0,Y 646.717,Z 1056.896,A -85,B 0,C 180,E1 6321.436,E2 6321.436} C_VEL
LIN {X 0,Y 648.53,Z 1023.083,A -85,B 0,C 180,E1 6323.424,E2 6323.424} C_VEL
LIN {X 0,Y 650.166,Z 985.974,A -85,B 0,C 180,E1 6324.989,E2 6324.989} C_VEL
LIN {X 0,Y 650.461,Z 952.967,A -85,B 0,C 180,E1 6325.962,E2 6325.962} C_VEL
LIN {X 0,Y 643.88,Z 933.758,A -85,B 0,C 180,E1 6326.593,E2 6326.593} C_VEL
LIN {X 0,Y 639.404,Z 927.122,A -85,B 0,C 180,E1 6327.01,E2 6327.01} C_VEL
LIN {X 0,Y 633.693,Z 923.44,A -85,B 0,C 180,E1 6327.788,E2 6327.788} C_VEL
LIN {X 0,Y 632.781,Z 923.03,A -85,B 0,C 180,E1 6328.198,E2 6328.198} C_VEL
LIN {X 0,Y 632.77,Z 923.03,A -85,B 0,C 180,E1 6333.328,E2 6333.328} C_VEL
LIN {X 0,Y 632.581,Z 923.03,A -85,B 0,C 180,E1 6338.393,E2 6338.393} C_VEL
LIN {X 0,Y 632.536,Z 923.03,A -85,B 0,C 180,E1 6344.241,E2 6344.241} C_VEL
LIN {X 0,Y 632.606,Z 923.03,A -85,B 0,C 180,E1 6349.859,E2 6349.859} C_VEL
LIN {X 0,Y 632.729,Z 923.03,A -85,B 0,C 180,E1 6355.047,E2 6355.047} C_VEL
LIN {X 0,Y 632.668,Z 923.03,A -85,B 0,C 180,E1 6359.913,E2 6359.913} C_VEL
LIN {X 0,Y 632.703,Z 923.03,A -85,B 0,C 180,E1 6362.086,E2 6362.086} C_VEL
LIN {X 0,Y 644.388,Z 956.989,A -85,B 0,C 180,E1 6362.952,E2 6362.952} C_VEL
LIN {X 0,Y 643.713,Z 1004.609,A -85,B 0,C 180,E1 6363.668,E2 6363.668} C_VEL
LIN {X 0,Y 642.39,Z 1044.389,A -85,B 0,C 180,E1 6364.783,E2 6364.783} C_VEL
LIN {X 0,Y 640.66,Z 1082.115,A -85,B 0,C 180,E1 6366.376,E2 6366.376} C_VEL
LIN {X 0,Y 638.886,Z 1116.908,A -85,B 0,C 180,E1 6368.417,E2 6368.417} C_VEL
LIN {X 0,Y 637.098,Z 1148.869,A -85,B 0,C 180,E1 6370.923,E2 6370.923} C_VEL
LIN {X 0,Y 635.623,Z 1176.799,A -85,B 0,C 180,E1 6373.832,E2 6373.832} C_VEL
LIN {X 0,Y 634.422,Z 1199.644,A -85,B 0,C 180,E1 6377.129,E2 6377.129} C_VEL
LIN {X 0,Y 633.811,Z 1216.036,A -85,B 0,C 180,E1 6380.406,E2 6380.406} C_VEL
LIN {X 0,Y 633.59,Z 1227.606,A -85,B 0,C 180,E1 6383.852,E2 6383.852} C_VEL
LIN {X 0,Y 633.509,Z 1233.919,A -85,B 0,C 180,E1 6387.278,E2 6387.278} C_VEL
LIN {X 0,Y 633.495,Z 1235.5,A -85,B 0,C 180,E1 6390.012,E2 6390.012} C_VEL
LIN {X 0,Y 633.525,Z 1233.891,A -85,B 0,C 180,E1 6392.746,E2 6392.746} C_VEL
LIN {X 0,Y 633.615,Z 1227.542,A -85,B 0,C 180,E1 6396.172,E2 6396.172} C_VEL
LIN {X 0,Y 633.834,Z 1215.931,A -85,B 0,C 180,E1 6399.618,E2 6399.618} C_VEL
LIN {X 0,Y 634.477,Z 1198.324,A -85,B 0,C 180,E1 6403.087,E2 6403.087} C_VEL
LIN {X 0,Y 635.582,Z 1176.703,A -85,B 0,C 180,E1 6406.18,E2 6406.18} C_VEL
LIN {X 0,Y 637.139,Z 1149.008,A -85,B 0,C 180,E1 6409.095,E2 6409.095} C_VEL
LIN {X 0,Y 638.97,Z 1117.546,A -85,B 0,C 180,E1 6411.605,E2 6411.605} C_VEL
LIN {X 0,Y 640.9,Z 1083.714,A -85,B 0,C 180,E1 6413.64,E2 6413.64} C_VEL
LIN {X 0,Y 642.754,Z 1046.477,A -85,B 0,C 180,E1 6415.269,E2 6415.269} C_VEL
LIN {X 0,Y 644.201,Z 1006.586,A -85,B 0,C 180,E1 6416.431,E2 6416.431} C_VEL
LIN {X 0,Y 645.172,Z 960.056,A -85,B 0,C 180,E1 6417.156,E2 6417.156} C_VEL
LIN {X 0,Y 642.185,Z 949.651,A -85,B 0,C 180,E1 6417.41,E2 6417.41} C_VEL
LIN {X 0,Y 632.74,Z 923.03,A -85,B 0,C 180,E1 6418.211,E2 6418.211} C_VEL
LIN {X 0,Y 632.776,Z 923.03,A -85,B 0,C 180,E1 6423.327,E2 6423.327} C_VEL
LIN {X 0,Y 632.635,Z 923.03,A -85,B 0,C 180,E1 6428.403,E2 6428.403} C_VEL
LIN {X 0,Y 632.56,Z 923.03,A -85,B 0,C 180,E1 6434.223,E2 6434.223} C_VEL
LIN {X 0,Y 632.576,Z 923.03,A -85,B 0,C 180,E1 6439.867,E2 6439.867} C_VEL
LIN {X 0,Y 632.691,Z 923.03,A -85,B 0,C 180,E1 6445.028,E2 6445.028} C_VEL
LIN {X 0,Y 632.697,Z 923.03,A -85,B 0,C 180,E1 6449.899,E2 6449.899} C_VEL
LIN {X 0,Y 632.853,Z 923.03,A -85,B 0,C 180,E1 6455.158,E2 6455.158} C_VEL
LIN {X 0,Y 632.814,Z 923.03,A -85,B 0,C 180,E1 6460.471,E2 6460.471} C_VEL
LIN {X 0,Y 632.897,Z 923.03,A -85,B 0,C 180,E1 6466.188,E2 6466.188} C_VEL
LIN {X 0,Y 633.142,Z 923.03,A -85,B 0,C 180,E1 6470.384,E2 6470.384} C_VEL
LIN {X 0,Y 633.148,Z 923.71,A -85,B 0,C 180,E1 6475.623,E2 6475.623} C_VEL
LIN {X 0,Y 636.748,Z 946.34,A -85,B 0,C 180,E1 6475.978,E2 6475.978} C_VEL
LIN {X 0,Y 636.708,Z 980.351,A -85,B 0,C 180,E1 6476.529,E2 6476.529} C_VEL
LIN {X 0,Y 636.281,Z 1009.233,A -85,B 0,C 180,E1 6477.534,E2 6477.534} C_VEL
LIN {X 0,Y 635.719,Z 1035.377,A -85,B 0,C 180,E1 6479.065,E2 6479.065} C_VEL
LIN {X 0,Y 635.138,Z 1057.18,A -85,B 0,C 180,E1 6481.001,E2 6481.001} C_VEL
LIN {X 0,Y 634.658,Z 1073.981,A -85,B 0,C 180,E1 6483.243,E2 6483.243} C_VEL
LIN {X 0,Y 634.205,Z 1085.938,A -85,B 0,C 180,E1 6485.813,E2 6485.813} C_VEL
LIN {X 0,Y 634.029,Z 1091.561,A -85,B 0,C 180,E1 6488.223,E2 6488.223} C_VEL
LIN {X 0,Y 633.979,Z 1092.139,A -85,B 0,C 180,E1 6490.994,E2 6490.994} C_VEL
LIN {X 0,Y 634.094,Z 1088.382,A -85,B 0,C 180,E1 6493.086,E2 6493.086} C_VEL
LIN {X 0,Y 634.374,Z 1078.779,A -85,B 0,C 180,E1 6495.658,E2 6495.658} C_VEL
LIN {X 0,Y 634.79,Z 1063.714,A -85,B 0,C 180,E1 6498.028,E2 6498.028} C_VEL
LIN {X 0,Y 635.369,Z 1043.748,A -85,B 0,C 180,E1 6500.092,E2 6500.092} C_VEL
LIN {X 0,Y 635.945,Z 1019.356,A -85,B 0,C 180,E1 6501.791,E2 6501.791} C_VEL
LIN {X 0,Y 636.547,Z 991.636,A -85,B 0,C 180,E1 6503.021,E2 6503.021} C_VEL
LIN {X 0,Y 636.769,Z 963.322,A -85,B 0,C 180,E1 6503.712,E2 6503.712} C_VEL
LIN {X 0,Y 635.865,Z 936.906,A -85,B 0,C 180,E1 6504.059,E2 6504.059} C_VEL
LIN {X 0,Y 633.032,Z 923.03,A -85,B 0,C 180,E1 6504.354,E2 6504.354} C_VEL
LIN {X 0,Y 632.654,Z 923.03,A -85,B 0,C 180,E1 6510.107,E2 6510.107} C_VEL
LIN {X 0,Y 632.637,Z 923.03,A -85,B 0,C 180,E1 6515.684,E2 6515.684} C_VEL
LIN {X 0,Y 632.595,Z 923.03,A -85,B 0,C 180,E1 6520.164,E2 6520.164} C_VEL
LIN {X 0,Y 632.558,Z 923.03,A -85,B 0,C 180,E1 6526.139,E2 6526.139} C_VEL
LIN {X 0,Y 632.692,Z 923.03,A -85,B 0,C 180,E1 6532.016,E2 6532.016} C_VEL
LIN {X 0,Y 632.665,Z 923.03,A -85,B 0,C 180,E1 6536.719,E2 6536.719} C_VEL
LIN {X 0,Y 632.817,Z 923.03,A -85,B 0,C 180,E1 6542.073,E2 6542.073} C_VEL
LIN {X 0,Y 632.87,Z 923.03,A -85,B 0,C 180,E1 6547.53,E2 6547.53} C_VEL
LIN {X 0,Y 632.99,Z 923.03,A -85,B 0,C 180,E1 6552.731,E2 6552.731} C_VEL
LIN {X 0,Y 633.008,Z 923.03,A -85,B 0,C 180,E1 6558.171,E2 6558.171} C_VEL
LIN {X 0,Y 633.228,Z 923.03,A -85,B 0,C 180,E1 6563.136,E2 6563.136} C_VEL
LIN {X 0,Y 633.307,Z 923.03,A -85,B 0,C 180,E1 6568.621,E2 6568.621} C_VEL
LIN {X 0,Y 633.269,Z 923.03,A -85,B 0,C 180,E1 6572.723,E2 6572.723} C_VEL
LIN {X 0,Y 633.179,Z 923.03,A -85,B 0,C 180,E1 6576.84,E2 6576.84} C_VEL
LIN {X 0,Y 633.075,Z 923.03,A -85,B 0,C 180,E1 6582.392,E2 6582.392} C_VEL
LIN {X 0,Y 633.01,Z 923.03,A -85,B 0,C 180,E1 6588.065,E2 6588.065} C_VEL
LIN {X 0,Y 632.876,Z 923.03,A -85,B 0,C 180,E1 6592.444,E2 6592.444} C_VEL
LIN {X 0,Y 632.839,Z 923.03,A -85,B 0,C 180,E1 6597.931,E2 6597.931} C_VEL
LIN {X 0,Y 632.782,Z 923.03,A -85,B 0,C 180,E1 6603.297,E2 6603.297} C_VEL
LIN {X 0,Y 632.625,Z 923.03,A -85,B 0,C 180,E1 6608.372,E2 6608.372} C_VEL
LIN {X 0,Y 632.75,Z 923.03,A -85,B 0,C 180,E1 6614.236,E2 6614.236} C_VEL
LIN {X 0,Y 632.654,Z 923.03,A -85,B 0,C 180,E1 6619.84,E2 6619.84} C_VEL
LIN {X 0,Y 632.6,Z 923.03,A -85,B 0,C 180,E1 6625.018,E2 6625.018} C_VEL
LIN {X 0,Y 632.705,Z 923.03,A -85,B 0,C 180,E1 6629.896,E2 6629.896} C_VEL
LIN {X 0,Y 632.94,Z 923.144,A -85,B 0,C 180,E1 6632.561,E2 6632.561} C_VEL
LIN {X 0,Y 644.138,Z 958.451,A -85,B 0,C 180,E1 6633.753,E2 6633.753} C_VEL
LIN {X 0,Y 642.501,Z 997.98,A -85,B 0,C 180,E1 6635.046,E2 6635.046} C_VEL
LIN {X 0,Y 640.591,Z 1034.733,A -85,B 0,C 180,E1 6636.821,E2 6636.821} C_VEL
LIN {X 0,Y 638.496,Z 1069.119,A -85,B 0,C 180,E1 6639.106,E2 6639.106} C_VEL
LIN {X 0,Y 636.556,Z 1100.17,A -85,B 0,C 180,E1 6641.886,E2 6641.886} C_VEL
LIN {X 0,Y 635.169,Z 1126.033,A -85,B 0,C 180,E1 6645.004,E2 6645.004} C_VEL
LIN {X 0,Y 634.227,Z 1146.393,A -85,B 0,C 180,E1 6648.314,E2 6648.314} C_VEL
LIN {X 0,Y 633.763,Z 1161.393,A -85,B 0,C 180,E1 6651.774,E2 6651.774} C_VEL
LIN {X 0,Y 633.546,Z 1170.804,A -85,B 0,C 180,E1 6655.21,E2 6655.21} C_VEL
LIN {X 0,Y 633.456,Z 1175.125,A -85,B 0,C 180,E1 6658.632,E2 6658.632} C_VEL
LIN {X 0,Y 633.458,Z 1175.06,A -85,B 0,C 180,E1 6661.365,E2 6661.365} C_VEL
LIN {X 0,Y 633.572,Z 1170.644,A -85,B 0,C 180,E1 6664.787,E2 6664.787} C_VEL
LIN {X 0,Y 633.762,Z 1161.1,A -85,B 0,C 180,E1 6668.223,E2 6668.223} C_VEL
LIN {X 0,Y 634.229,Z 1145.951,A -85,B 0,C 180,E1 6671.683,E2 6671.683} C_VEL
LIN {X 0,Y 635.128,Z 1125.432,A -85,B 0,C 180,E1 6674.994,E2 6674.994} C_VEL
LIN {X 0,Y 636.614,Z 1099.359,A -85,B 0,C 180,E1 6678.11,E2 6678.11} C_VEL
LIN {X 0,Y 638.425,Z 1069.082,A -85,B 0,C 180,E1 6680.794,E2 6680.794} C_VEL
LIN {X 0,Y 640.412,Z 1036.19,A -85,B 0,C 180,E1 6682.971,E2 6682.971} C_VEL
LIN {X 0,Y 642.131,Z 1000.796,A -85,B 0,C 180,E1 6684.688,E2 6684.688} C_VEL
LIN {X 0,Y 643.552,Z 963.407,A -85,B 0,C 180,E1 6685.937,E2 6685.937} C_VEL
LIN {X 0,Y 642.899,Z 954.454,A -85,B 0,C 180,E1 6686.197,E2 6686.197} C_VEL
LIN {X 0,Y 632.858,Z 923.03,A -85,B 0,C 180,E1 6687.194,E2 6687.194} C_VEL
LIN {X 0,Y 632.781,Z 923.03,A -85,B 0,C 180,E1 6688.198,E2 6688.198} C_VEL
LIN {X 0,Y 631.516,Z 923.03,A -85,B 0,C 180,E1 6688.982,E2 6688.982} C_VEL
LIN {X 0,Y 624.901,Z 923.03,A -85,B 0,C 180,E1 6691.111,E2 6691.111} C_VEL
LIN {X 0,Y 624.806,Z 923.03,A -85,B 0,C 180,E1 6691.313,E2 6691.313} C_VEL
LIN {X 0,Y 624.748,Z 923.03,A -85,B 0,C 180,E1 6695.484,E2 6695.484} C_VEL
LIN {X 0,Y 624.615,Z 923.03,A -85,B 0,C 180,E1 6701.437,E2 6701.437} C_VEL
LIN {X 0,Y 624.601,Z 923.03,A -85,B 0,C 180,E1 6706.532,E2 6706.532} C_VEL
LIN {X 0,Y 624.658,Z 923.03,A -85,B 0,C 180,E1 6711.047,E2 6711.047} C_VEL
LIN {X 0,Y 624.768,Z 923.03,A -85,B 0,C 180,E1 6716.219,E2 6716.219} C_VEL
LIN {X 0,Y 624.78,Z 923.03,A -85,B 0,C 180,E1 6721.751,E2 6721.751} C_VEL
LIN {X 0,Y 637.093,Z 961.153,A -85,B 0,C 180,E1 6722.741,E2 6722.741} C_VEL
LIN {X 0,Y 636.292,Z 1005.056,A -85,B 0,C 180,E1 6723.432,E2 6723.432} C_VEL
LIN {X 0,Y 634.872,Z 1044.374,A -85,B 0,C 180,E1 6724.554,E2 6724.554} C_VEL
LIN {X 0,Y 633.109,Z 1081.953,A -85,B 0,C 180,E1 6726.165,E2 6726.165} C_VEL
LIN {X 0,Y 631.218,Z 1116.823,A -85,B 0,C 180,E1 6728.234,E2 6728.234} C_VEL
LIN {X 0,Y 629.339,Z 1148.404,A -85,B 0,C 180,E1 6730.737,E2 6730.737} C_VEL
LIN {X 0,Y 627.792,Z 1176.777,A -85,B 0,C 180,E1 6733.724,E2 6733.724} C_VEL
LIN {X 0,Y 626.61,Z 1199.493,A -85,B 0,C 180,E1 6736.947,E2 6736.947} C_VEL
LIN {X 0,Y 625.956,Z 1216.036,A -85,B 0,C 180,E1 6740.284,E2 6740.284} C_VEL
LIN {X 0,Y 625.698,Z 1227.607,A -85,B 0,C 180,E1 6743.774,E2 6743.774} C_VEL
LIN {X 0,Y 625.605,Z 1233.918,A -85,B 0,C 180,E1 6747.244,E2 6747.244} C_VEL
LIN {X 0,Y 625.595,Z 1235.5,A -85,B 0,C 180,E1 6750.012,E2 6750.012} C_VEL
LIN {X 0,Y 625.621,Z 1233.891,A -85,B 0,C 180,E1 6752.781,E2 6752.781} C_VEL
LIN {X 0,Y 625.722,Z 1227.542,A -85,B 0,C 180,E1 6756.251,E2 6756.251} C_VEL
LIN {X 0,Y 625.975,Z 1215.931,A -85,B 0,C 180,E1 6759.74,E2 6759.74} C_VEL
LIN {X 0,Y 626.643,Z 1198.24,A -85,B 0,C 180,E1 6763.254,E2 6763.254} C_VEL
LIN {X 0,Y 627.847,Z 1175.435,A -85,B 0,C 180,E1 6766.462,E2 6766.462} C_VEL
LIN {X 0,Y 629.421,Z 1148.836,A -85,B 0,C 180,E1 6769.286,E2 6769.286} C_VEL
LIN {X 0,Y 631.457,Z 1116.685,A -85,B 0,C 180,E1 6771.876,E2 6771.876} C_VEL
LIN {X 0,Y 633.519,Z 1082.675,A -85,B 0,C 180,E1 6773.933,E2 6773.933} C_VEL
LIN {X 0,Y 635.401,Z 1046.141,A -85,B 0,C 180,E1 6775.545,E2 6775.545} C_VEL
LIN {X 0,Y 636.926,Z 1006.713,A -85,B 0,C 180,E1 6776.709,E2 6776.709} C_VEL
LIN {X 0,Y 637.748,Z 958.763,A -85,B 0,C 180,E1 6777.475,E2 6777.475} C_VEL
LIN {X 0,Y 624.862,Z 923.03,A -85,B 0,C 180,E1 6778.552,E2 6778.552} C_VEL
LIN {X 0,Y 624.805,Z 923.03,A -85,B 0,C 180,E1 6783.808,E2 6783.808} C_VEL
LIN {X 0,Y 624.626,Z 923.03,A -85,B 0,C 180,E1 6789.275,E2 6789.275} C_VEL
LIN {X 0,Y 624.62,Z 923.03,A -85,B 0,C 180,E1 6794.565,E2 6794.565} C_VEL
LIN {X 0,Y 624.6,Z 923.03,A -85,B 0,C 180,E1 6799.218,E2 6799.218} C_VEL
LIN {X 0,Y 624.779,Z 923.03,A -85,B 0,C 180,E1 6804.518,E2 6804.518} C_VEL
LIN {X 0,Y 624.785,Z 923.03,A -85,B 0,C 180,E1 6809.477,E2 6809.477} C_VEL
LIN {X 0,Y 624.893,Z 923.03,A -85,B 0,C 180,E1 6814.199,E2 6814.199} C_VEL
LIN {X 0,Y 624.952,Z 923.03,A -85,B 0,C 180,E1 6818.736,E2 6818.736} C_VEL
LIN {X 0,Y 624.893,Z 923.03,A -85,B 0,C 180,E1 6824.575,E2 6824.575} C_VEL
LIN {X 0,Y 625.243,Z 923.03,A -85,B 0,C 180,E1 6830.262,E2 6830.262} C_VEL
LIN {X 0,Y 625.2,Z 923.03,A -85,B 0,C 180,E1 6835.409,E2 6835.409} C_VEL
LIN {X 0,Y 629.075,Z 944.581,A -85,B 0,C 180,E1 6835.783,E2 6835.783} C_VEL
LIN {X 0,Y 629.055,Z 981.324,A -85,B 0,C 180,E1 6836.374,E2 6836.374} C_VEL
LIN {X 0,Y 628.604,Z 1010.78,A -85,B 0,C 180,E1 6837.418,E2 6837.418} C_VEL
LIN {X 0,Y 628,Z 1036.771,A -85,B 0,C 180,E1 6838.967,E2 6838.967} C_VEL
LIN {X 0,Y 627.401,Z 1058.095,A -85,B 0,C 180,E1 6840.891,E2 6840.891} C_VEL
LIN {X 0,Y 626.896,Z 1074.6,A -85,B 0,C 180,E1 6843.11,E2 6843.11} C_VEL
LIN {X 0,Y 626.412,Z 1086.106,A -85,B 0,C 180,E1 6845.539,E2 6845.539} C_VEL
LIN {X 0,Y 626.258,Z 1091.592,A -85,B 0,C 180,E1 6847.615,E2 6847.615} C_VEL
LIN {X 0,Y 626.172,Z 1093.557,A -85,B 0,C 180,E1 6849.727,E2 6849.727} C_VEL
LIN {X 0,Y 626.192,Z 1092.254,A -85,B 0,C 180,E1 6851.696,E2 6851.696} C_VEL
LIN {X 0,Y 626.386,Z 1085.834,A -85,B 0,C 180,E1 6854.277,E2 6854.277} C_VEL
LIN {X 0,Y 626.676,Z 1073.537,A -85,B 0,C 180,E1 6856.821,E2 6856.821} C_VEL
LIN {X 0,Y 627.155,Z 1057.167,A -85,B 0,C 180,E1 6858.984,E2 6858.984} C_VEL
LIN {X 0,Y 627.874,Z 1035.325,A -85,B 0,C 180,E1 6860.937,E2 6860.937} C_VEL
LIN {X 0,Y 628.52,Z 1010.242,A -85,B 0,C 180,E1 6862.434,E2 6862.434} C_VEL
LIN {X 0,Y 628.966,Z 982.037,A -85,B 0,C 180,E1 6863.482,E2 6863.482} C_VEL
LIN {X 0,Y 629.11,Z 949.26,A -85,B 0,C 180,E1 6864.054,E2 6864.054} C_VEL
LIN {X 0,Y 626.617,Z 930.618,A -85,B 0,C 180,E1 6864.333,E2 6864.333} C_VEL
LIN {X 0,Y 625.136,Z 923.03,A -85,B 0,C 180,E1 6864.52,E2 6864.52} C_VEL
LIN {X 0,Y 624.753,Z 923.03,A -85,B 0,C 180,E1 6870.528,E2 6870.528} C_VEL
LIN {X 0,Y 624.728,Z 923.03,A -85,B 0,C 180,E1 6875.489,E2 6875.489} C_VEL
LIN {X 0,Y 624.597,Z 923.03,A -85,B 0,C 180,E1 6880.786,E2 6880.786} C_VEL
LIN {X 0,Y 624.618,Z 923.03,A -85,B 0,C 180,E1 6886.535,E2 6886.535} C_VEL
LIN {X 0,Y 624.705,Z 923.03,A -85,B 0,C 180,E1 6891.019,E2 6891.019} C_VEL
LIN {X 0,Y 624.695,Z 923.03,A -85,B 0,C 180,E1 6896.185,E2 6896.185} C_VEL
LIN {X 0,Y 624.835,Z 923.03,A -85,B 0,C 180,E1 6901.063,E2 6901.063} C_VEL
LIN {X 0,Y 624.979,Z 923.03,A -85,B 0,C 180,E1 6905.719,E2 6905.719} C_VEL
LIN {X 0,Y 625.072,Z 923.03,A -85,B 0,C 180,E1 6910.534,E2 6910.534} C_VEL
LIN {X 0,Y 625.013,Z 923.03,A -85,B 0,C 180,E1 6915.998,E2 6915.998} C_VEL
LIN {X 0,Y 625.273,Z 923.03,A -85,B 0,C 180,E1 6921.651,E2 6921.651} C_VEL
LIN {X 0,Y 625.533,Z 923.03,A -85,B 0,C 180,E1 6927.219,E2 6927.219} C_VEL
LIN {X 0,Y 625.367,Z 923.03,A -85,B 0,C 180,E1 6932.758,E2 6932.758} C_VEL
LIN {X 0,Y 625.242,Z 923.03,A -85,B 0,C 180,E1 6937.726,E2 6937.726} C_VEL
LIN {X 0,Y 625.156,Z 923.03,A -85,B 0,C 180,E1 6942.551,E2 6942.551} C_VEL
LIN {X 0,Y 625.135,Z 923.03,A -85,B 0,C 180,E1 6946.848,E2 6946.848} C_VEL
LIN {X 0,Y 625.004,Z 923.03,A -85,B 0,C 180,E1 6951.249,E2 6951.249} C_VEL
LIN {X 0,Y 624.893,Z 923.03,A -85,B 0,C 180,E1 6956.524,E2 6956.524} C_VEL
LIN {X 0,Y 624.863,Z 923.03,A -85,B 0,C 180,E1 6962.175,E2 6962.175} C_VEL
LIN {X 0,Y 624.729,Z 923.03,A -85,B 0,C 180,E1 6967.188,E2 6967.188} C_VEL
LIN {X 0,Y 624.804,Z 923.03,A -85,B 0,C 180,E1 6972.602,E2 6972.602} C_VEL
LIN {X 0,Y 624.722,Z 923.03,A -85,B 0,C 180,E1 6977.367,E2 6977.367} C_VEL
LIN {X 0,Y 624.709,Z 923.03,A -85,B 0,C 180,E1 6982.934,E2 6982.934} C_VEL
LIN {X 0,Y 624.771,Z 923.03,A -85,B 0,C 180,E1 6987.851,E2 6987.851} C_VEL
LIN {X 0,Y 624.994,Z 923.03,A -85,B 0,C 180,E1 6992.211,E2 6992.211} C_VEL
LIN {X 0,Y 636.898,Z 960.067,A -85,B 0,C 180,E1 6993.508,E2 6993.508} C_VEL
LIN {X 0,Y 635.183,Z 998.237,A -85,B 0,C 180,E1 6994.776,E2 6994.776} C_VEL
LIN {X 0,Y 633.21,Z 1034.084,A -85,B 0,C 180,E1 6996.518,E2 6996.518} C_VEL
LIN {X 0,Y 631.015,Z 1067.887,A -85,B 0,C 180,E1 6998.763,E2 6998.763} C_VEL
LIN {X 0,Y 629.054,Z 1098.465,A -85,B 0,C 180,E1 7001.484,E2 7001.484} C_VEL
LIN {X 0,Y 627.493,Z 1124.915,A -85,B 0,C 180,E1 7004.638,E2 7004.638} C_VEL
LIN {X 0,Y 626.442,Z 1144.665,A -85,B 0,C 180,E1 7007.824,E2 7007.824} C_VEL
LIN {X 0,Y 625.912,Z 1160.213,A -85,B 0,C 180,E1 7011.32,E2 7011.32} C_VEL
LIN {X 0,Y 625.674,Z 1170.801,A -85,B 0,C 180,E1 7015.149,E2 7015.149} C_VEL
LIN {X 0,Y 625.554,Z 1175.125,A -85,B 0,C 180,E1 7018.614,E2 7018.614} C_VEL
LIN {X 0,Y 625.557,Z 1175.06,A -85,B 0,C 180,E1 7021.383,E2 7021.383} C_VEL
LIN {X 0,Y 625.7,Z 1170.643,A -85,B 0,C 180,E1 7024.847,E2 7024.847} C_VEL
LIN {X 0,Y 625.869,Z 1161.1,A -85,B 0,C 180,E1 7028.328,E2 7028.328} C_VEL
LIN {X 0,Y 626.402,Z 1146.033,A -85,B 0,C 180,E1 7031.814,E2 7031.814} C_VEL
LIN {X 0,Y 627.379,Z 1125.59,A -85,B 0,C 180,E1 7035.183,E2 7035.183} C_VEL
LIN {X 0,Y 628.95,Z 1099.64,A -85,B 0,C 180,E1 7038.304,E2 7038.304} C_VEL
LIN {X 0,Y 630.808,Z 1070.278,A -85,B 0,C 180,E1 7040.942,E2 7040.942} C_VEL
LIN {X 0,Y 632.879,Z 1037.279,A -85,B 0,C 180,E1 7043.16,E2 7043.16} C_VEL
LIN {X 0,Y 634.696,Z 1001.878,A -85,B 0,C 180,E1 7044.903,E2 7044.903} C_VEL
LIN {X 0,Y 636.192,Z 964.359,A -85,B 0,C 180,E1 7046.178,E2 7046.178} C_VEL
LIN {X 0,Y 635.168,Z 955.355,A -85,B 0,C 180,E1 7046.458,E2 7046.458} C_VEL
LIN {X 0,Y 624.939,Z 923.03,A -85,B 0,C 180,E1 7047.581,E2 7047.581} C_VEL
LIN {X 0,Y 624.806,Z 923.03,A -85,B 0,C 180,E1 7051.313,E2 7051.313} C_VEL
LIN {X 0,Y 620.898,Z 923.03,A -85,B 0,C 180,E1 7052.881,E2 7052.881} C_VEL
LIN {X 0,Y 616.843,Z 923.03,A -85,B 0,C 180,E1 7054.469,E2 7054.469} C_VEL
LIN {X 0,Y 616.712,Z 923.03,A -85,B 0,C 180,E1 7059.571,E2 7059.571} C_VEL
LIN {X 0,Y 616.694,Z 923.03,A -85,B 0,C 180,E1 7065.281,E2 7065.281} C_VEL
LIN {X 0,Y 616.745,Z 923.03,A -85,B 0,C 180,E1 7070.45,E2 7070.45} C_VEL
LIN {X 0,Y 616.879,Z 923.03,A -85,B 0,C 180,E1 7075.727,E2 7075.727} C_VEL
LIN {X 0,Y 616.86,Z 923.03,A -85,B 0,C 180,E1 7081.422,E2 7081.422} C_VEL
LIN {X 0,Y 629.687,Z 960.667,A -85,B 0,C 180,E1 7082.458,E2 7082.458} C_VEL
LIN {X 0,Y 628.867,Z 1005.713,A -85,B 0,C 180,E1 7083.192,E2 7083.192} C_VEL
LIN {X 0,Y 627.336,Z 1045.562,A -85,B 0,C 180,E1 7084.363,E2 7084.363} C_VEL
LIN {X 0,Y 625.374,Z 1084.211,A -85,B 0,C 180,E1 7086.069,E2 7086.069} C_VEL
LIN {X 0,Y 623.337,Z 1120.623,A -85,B 0,C 180,E1 7088.319,E2 7088.319} C_VEL
LIN {X 0,Y 621.276,Z 1153.06,A -85,B 0,C 180,E1 7091.03,E2 7091.03} C_VEL
LIN {X 0,Y 619.725,Z 1179.619,A -85,B 0,C 180,E1 7093.982,E2 7093.982} C_VEL
LIN {X 0,Y 618.691,Z 1200.863,A -85,B 0,C 180,E1 7097.136,E2 7097.136} C_VEL
LIN {X 0,Y 618.059,Z 1217.304,A -85,B 0,C 180,E1 7100.514,E2 7100.514} C_VEL
LIN {X 0,Y 617.821,Z 1227.606,A -85,B 0,C 180,E1 7103.694,E2 7103.694} C_VEL
LIN {X 0,Y 617.721,Z 1233.917,A -85,B 0,C 180,E1 7107.208,E2 7107.208} C_VEL
LIN {X 0,Y 617.705,Z 1235.5,A -85,B 0,C 180,E1 7110.012,E2 7110.012} C_VEL
LIN {X 0,Y 617.737,Z 1233.89,A -85,B 0,C 180,E1 7112.816,E2 7112.816} C_VEL
LIN {X 0,Y 617.843,Z 1227.542,A -85,B 0,C 180,E1 7116.331,E2 7116.331} C_VEL
LIN {X 0,Y 618.101,Z 1215.801,A -85,B 0,C 180,E1 7119.865,E2 7119.865} C_VEL
LIN {X 0,Y 618.791,Z 1197.703,A -85,B 0,C 180,E1 7123.426,E2 7123.426} C_VEL
LIN {X 0,Y 620.09,Z 1175.014,A -85,B 0,C 180,E1 7126.65,E2 7126.65} C_VEL
LIN {X 0,Y 621.741,Z 1148.105,A -85,B 0,C 180,E1 7129.534,E2 7129.534} C_VEL
LIN {X 0,Y 623.836,Z 1117.113,A -85,B 0,C 180,E1 7132.063,E2 7132.063} C_VEL
LIN {X 0,Y 626.034,Z 1082.982,A -85,B 0,C 180,E1 7134.163,E2 7134.163} C_VEL
LIN {X 0,Y 628.046,Z 1046.049,A -85,B 0,C 180,E1 7135.818,E2 7135.818} C_VEL
LIN {X 0,Y 629.682,Z 1006.838,A -85,B 0,C 180,E1 7136.993,E2 7136.993} C_VEL
LIN {X 0,Y 630.652,Z 960.862,A -85,B 0,C 180,E1 7137.745,E2 7137.745} C_VEL
LIN {X 0,Y 616.923,Z 923.03,A -85,B 0,C 180,E1 7138.882,E2 7138.882} C_VEL
LIN {X 0,Y 616.879,Z 923.03,A -85,B 0,C 180,E1 7144.303,E2 7144.303} C_VEL
LIN {X 0,Y 616.701,Z 923.03,A -85,B 0,C 180,E1 7149.586,E2 7149.586} C_VEL
LIN {X 0,Y 616.73,Z 923.03,A -85,B 0,C 180,E1 7155.292,E2 7155.292} C_VEL
LIN {X 0,Y 616.714,Z 923.03,A -85,B 0,C 180,E1 7160.429,E2 7160.429} C_VEL
LIN {X 0,Y 616.837,Z 923.03,A -85,B 0,C 180,E1 7165.708,E2 7165.708} C_VEL
LIN {X 0,Y 616.865,Z 923.03,A -85,B 0,C 180,E1 7170.666,E2 7170.666} C_VEL
LIN {X 0,Y 616.991,Z 923.03,A -85,B 0,C 180,E1 7175.397,E2 7175.397} C_VEL
LIN {X 0,Y 616.98,Z 923.03,A -85,B 0,C 180,E1 7179.949,E2 7179.949} C_VEL
LIN {X 0,Y 617.05,Z 923.03,A -85,B 0,C 180,E1 7185.826,E2 7185.826} C_VEL
LIN {X 0,Y 617.323,Z 923.03,A -85,B 0,C 180,E1 7190.135,E2 7190.135} C_VEL
LIN {X 0,Y 617.304,Z 923.03,A -85,B 0,C 180,E1 7195.215,E2 7195.215} C_VEL
LIN {X 0,Y 621.462,Z 947.637,A -85,B 0,C 180,E1 7195.64,E2 7195.64} C_VEL
LIN {X 0,Y 621.437,Z 982.794,A -85,B 0,C 180,E1 7196.23,E2 7196.23} C_VEL
LIN {X 0,Y 620.92,Z 1012.33,A -85,B 0,C 180,E1 7197.299,E2 7197.299} C_VEL
LIN {X 0,Y 620.284,Z 1038.165,A -85,B 0,C 180,E1 7198.867,E2 7198.867} C_VEL
LIN {X 0,Y 619.612,Z 1059.736,A -85,B 0,C 180,E1 7200.857,E2 7200.857} C_VEL
LIN {X 0,Y 619.072,Z 1076.318,A -85,B 0,C 180,E1 7203.15,E2 7203.15} C_VEL
LIN {X 0,Y 618.604,Z 1087.519,A -85,B 0,C 180,E1 7205.609,E2 7205.609} C_VEL
LIN {X 0,Y 618.44,Z 1092.584,A -85,B 0,C 180,E1 7207.613,E2 7207.613} C_VEL
LIN {X 0,Y 618.334,Z 1094.511,A -85,B 0,C 180,E1 7209.851,E2 7209.851} C_VEL
LIN {X 0,Y 618.398,Z 1092.428,A -85,B 0,C 180,E1 7212.163,E2 7212.163} C_VEL
LIN {X 0,Y 618.608,Z 1085.216,A -85,B 0,C 180,E1 7214.718,E2 7214.718} C_VEL
LIN {X 0,Y 619.014,Z 1072.276,A -85,B 0,C 180,E1 7217.234,E2 7217.234} C_VEL
LIN {X 0,Y 619.53,Z 1054.891,A -85,B 0,C 180,E1 7219.412,E2 7219.412} C_VEL
LIN {X 0,Y 620.226,Z 1032.736,A -85,B 0,C 180,E1 7221.299,E2 7221.299} C_VEL
LIN {X 0,Y 620.898,Z 1006.641,A -85,B 0,C 180,E1 7222.774,E2 7222.774} C_VEL
LIN {X 0,Y 621.304,Z 977.788,A -85,B 0,C 180,E1 7223.755,E2 7223.755} C_VEL
LIN {X 0,Y 620.689,Z 939.893,A -85,B 0,C 180,E1 7224.348,E2 7224.348} C_VEL
LIN {X 0,Y 617.199,Z 923.03,A -85,B 0,C 180,E1 7224.706,E2 7224.706} C_VEL
LIN {X 0,Y 616.82,Z 923.03,A -85,B 0,C 180,E1 7230.963,E2 7230.963} C_VEL
LIN {X 0,Y 616.788,Z 923.03,A -85,B 0,C 180,E1 7236.038,E2 7236.038} C_VEL
LIN {X 0,Y 616.717,Z 923.03,A -85,B 0,C 180,E1 7241.421,E2 7241.421} C_VEL
LIN {X 0,Y 616.752,Z 923.03,A -85,B 0,C 180,E1 7247.312,E2 7247.312} C_VEL
LIN {X 0,Y 616.771,Z 923.03,A -85,B 0,C 180,E1 7252.218,E2 7252.218} C_VEL
LIN {X 0,Y 616.787,Z 923.03,A -85,B 0,C 180,E1 7257.374,E2 7257.374} C_VEL
LIN {X 0,Y 616.962,Z 923.03,A -85,B 0,C 180,E1 7262.255,E2 7262.255} C_VEL
LIN {X 0,Y 617.033,Z 923.03,A -85,B 0,C 180,E1 7266.92,E2 7266.92} C_VEL
LIN {X 0,Y 617.143,Z 923.03,A -85,B 0,C 180,E1 7272.737,E2 7272.737} C_VEL
LIN {X 0,Y 617.242,Z 923.03,A -85,B 0,C 180,E1 7278.694,E2 7278.694} C_VEL
LIN {X 0,Y 617.405,Z 923.03,A -85,B 0,C 180,E1 7284.37,E2 7284.37} C_VEL
LIN {X 0,Y 617.529,Z 923.03,A -85,B 0,C 180,E1 7288.586,E2 7288.586} C_VEL
LIN {X 0,Y 617.465,Z 923.03,A -85,B 0,C 180,E1 7292.793,E2 7292.793} C_VEL
LIN {X 0,Y 617.371,Z 923.03,A -85,B 0,C 180,E1 7297.016,E2 7297.016} C_VEL
LIN {X 0,Y 617.264,Z 923.03,A -85,B 0,C 180,E1 7302.714,E2 7302.714} C_VEL
LIN {X 0,Y 617.177,Z 923.03,A -85,B 0,C 180,E1 7307.273,E2 7307.273} C_VEL
LIN {X 0,Y 617.015,Z 923.03,A -85,B 0,C 180,E1 7313.054,E2 7313.054} C_VEL
LIN {X 0,Y 616.953,Z 923.03,A -85,B 0,C 180,E1 7318.143,E2 7318.143} C_VEL
LIN {X 0,Y 616.897,Z 923.03,A -85,B 0,C 180,E1 7323.606,E2 7323.606} C_VEL
LIN {X 0,Y 616.778,Z 923.03,A -85,B 0,C 180,E1 7329.548,E2 7329.548} C_VEL
LIN {X 0,Y 616.889,Z 923.03,A -85,B 0,C 180,E1 7334.733,E2 7334.733} C_VEL
LIN {X 0,Y 616.776,Z 923.03,A -85,B 0,C 180,E1 7340.43,E2 7340.43} C_VEL
LIN {X 0,Y 616.785,Z 923.03,A -85,B 0,C 180,E1 7346.376,E2 7346.376} C_VEL
LIN {X 0,Y 617.069,Z 923.03,A -85,B 0,C 180,E1 7351.857,E2 7351.857} C_VEL
LIN {X 0,Y 629.601,Z 962.52,A -85,B 0,C 180,E1 7353.279,E2 7353.279} C_VEL
LIN {X 0,Y 627.827,Z 999.596,A -85,B 0,C 180,E1 7354.546,E2 7354.546} C_VEL
LIN {X 0,Y 625.734,Z 1035.362,A -85,B 0,C 180,E1 7356.319,E2 7356.319} C_VEL
LIN {X 0,Y 623.452,Z 1068.867,A -85,B 0,C 180,E1 7358.586,E2 7358.586} C_VEL
LIN {X 0,Y 621.43,Z 1098.654,A -85,B 0,C 180,E1 7361.273,E2 7361.273} C_VEL
LIN {X 0,Y 619.783,Z 1125.026,A -85,B 0,C 180,E1 7364.442,E2 7364.442} C_VEL
LIN {X 0,Y 618.607,Z 1145.36,A -85,B 0,C 180,E1 7367.765,E2 7367.765} C_VEL
LIN {X 0,Y 618.026,Z 1160.27,A -85,B 0,C 180,E1 7371.208,E2 7371.208} C_VEL
LIN {X 0,Y 617.773,Z 1170.798,A -85,B 0,C 180,E1 7375.087,E2 7375.087} C_VEL
LIN {X 0,Y 617.669,Z 1175.125,A -85,B 0,C 180,E1 7378.597,E2 7378.597} C_VEL
LIN {X 0,Y 617.672,Z 1175.059,A -85,B 0,C 180,E1 7381.4,E2 7381.4} C_VEL
LIN {X 0,Y 617.799,Z 1170.642,A -85,B 0,C 180,E1 7384.909,E2 7384.909} C_VEL
LIN {X 0,Y 618.001,Z 1159.963,A -85,B 0,C 180,E1 7388.789,E2 7388.789} C_VEL
LIN {X 0,Y 618.644,Z 1144.139,A -85,B 0,C 180,E1 7392.384,E2 7392.384} C_VEL
LIN {X 0,Y 619.8,Z 1123.276,A -85,B 0,C 180,E1 7395.716,E2 7395.716} C_VEL
LIN {X 0,Y 621.33,Z 1099.04,A -85,B 0,C 180,E1 7398.595,E2 7398.595} C_VEL
LIN {X 0,Y 623.292,Z 1070.181,A -85,B 0,C 180,E1 7401.192,E2 7401.192} C_VEL
LIN {X 0,Y 625.402,Z 1037.796,A -85,B 0,C 180,E1 7403.385,E2 7403.385} C_VEL
LIN {X 0,Y 627.252,Z 1003.087,A -85,B 0,C 180,E1 7405.119,E2 7405.119} C_VEL
LIN {X 0,Y 628.86,Z 965.197,A -85,B 0,C 180,E1 7406.43,E2 7406.43} C_VEL
LIN {X 0,Y 627.697,Z 956.842,A -85,B 0,C 180,E1 7406.708,E2 7406.708} C_VEL
LIN {X 0,Y 617.039,Z 923.03,A -85,B 0,C 180,E1 7407.866,E2 7407.866} C_VEL
LIN {X 0,Y 616.93,Z 923.03,A -85,B 0,C 180,E1 7413.644,E2 7413.644} C_VEL
LIN {X 0,Y 616.843,Z 923.03,A -85,B 0,C 180,E1 7414.469,E2 7414.469} C_VEL
LIN {X 0,Y 612.756,Z 923.03,A -85,B 0,C 180,E1 7416.058,E2 7416.058} C_VEL
LIN {X 0,Y 608.786,Z 923.03,A -85,B 0,C 180,E1 7417.668,E2 7417.668} C_VEL
LIN {X 0,Y 608.804,Z 923.03,A -85,B 0,C 180,E1 7422.077,E2 7422.077} C_VEL
LIN {X 0,Y 608.817,Z 923.03,A -85,B 0,C 180,E1 7428.123,E2 7428.123} C_VEL
LIN {X 0,Y 608.884,Z 923.03,A -85,B 0,C 180,E1 7433.463,E2 7433.463} C_VEL
LIN {X 0,Y 608.911,Z 923.03,A -85,B 0,C 180,E1 7438.609,E2 7438.609} C_VEL
LIN {X 0,Y 608.959,Z 923.03,A -85,B 0,C 180,E1 7441.056,E2 7441.056} C_VEL
LIN {X 0,Y 622.317,Z 962.373,A -85,B 0,C 180,E1 7442.192,E2 7442.192} C_VEL
LIN {X 0,Y 621.446,Z 1007.007,A -85,B 0,C 180,E1 7442.956,E2 7442.956} C_VEL
LIN {X 0,Y 619.693,Z 1048.785,A -85,B 0,C 180,E1 7444.237,E2 7444.237} C_VEL
LIN {X 0,Y 617.595,Z 1088.08,A -85,B 0,C 180,E1 7446.068,E2 7446.068} C_VEL
LIN {X 0,Y 615.482,Z 1122.929,A -85,B 0,C 180,E1 7448.312,E2 7448.312} C_VEL
LIN {X 0,Y 613.44,Z 1153.846,A -85,B 0,C 180,E1 7450.965,E2 7450.965} C_VEL
LIN {X 0,Y 611.882,Z 1179.63,A -85,B 0,C 180,E1 7453.884,E2 7453.884} C_VEL
LIN {X 0,Y 610.792,Z 1201.214,A -85,B 0,C 180,E1 7457.149,E2 7457.149} C_VEL
LIN {X 0,Y 610.19,Z 1216.775,A -85,B 0,C 180,E1 7460.391,E2 7460.391} C_VEL
LIN {X 0,Y 609.944,Z 1227.312,A -85,B 0,C 180,E1 7463.612,E2 7463.612} C_VEL
LIN {X 0,Y 609.816,Z 1233.805,A -85,B 0,C 180,E1 7467.172,E2 7467.172} C_VEL
LIN {X 0,Y 609.805,Z 1235.428,A -85,B 0,C 180,E1 7470.013,E2 7470.013} C_VEL
LIN {X 0,Y 609.814,Z 1232.902,A -85,B 0,C 180,E1 7473.564,E2 7473.564} C_VEL
LIN {X 0,Y 609.969,Z 1225.309,A -85,B 0,C 180,E1 7477.127,E2 7477.127} C_VEL
LIN {X 0,Y 610.35,Z 1212.202,A -85,B 0,C 180,E1 7480.713,E2 7480.713} C_VEL
LIN {X 0,Y 611.178,Z 1193.841,A -85,B 0,C 180,E1 7484.143,E2 7484.143} C_VEL
LIN {X 0,Y 612.583,Z 1170.108,A -85,B 0,C 180,E1 7487.39,E2 7487.39} C_VEL
LIN {X 0,Y 614.628,Z 1139.955,A -85,B 0,C 180,E1 7490.469,E2 7490.469} C_VEL
LIN {X 0,Y 616.92,Z 1106.954,A -85,B 0,C 180,E1 7492.989,E2 7492.989} C_VEL
LIN {X 0,Y 619.265,Z 1071.392,A -85,B 0,C 180,E1 7495.008,E2 7495.008} C_VEL
LIN {X 0,Y 621.437,Z 1032.997,A -85,B 0,C 180,E1 7496.55,E2 7496.55} C_VEL
LIN {X 0,Y 622.945,Z 994.152,A -85,B 0,C 180,E1 7497.553,E2 7497.553} C_VEL
LIN {X 0,Y 622.895,Z 961.305,A -85,B 0,C 180,E1 7498.072,E2 7498.072} C_VEL
LIN {X 0,Y 609.017,Z 923.03,A -85,B 0,C 180,E1 7499.286,E2 7499.286} C_VEL
LIN {X 0,Y 608.918,Z 923.03,A -85,B 0,C 180,E1 7505.025,E2 7505.025} C_VEL
LIN {X 0,Y 608.803,Z 923.03,A -85,B 0,C 180,E1 7510.203,E2 7510.203} C_VEL
LIN {X 0,Y 608.778,Z 923.03,A -85,B 0,C 180,E1 7516.053,E2 7516.053} C_VEL
LIN {X 0,Y 608.846,Z 923.03,A -85,B 0,C 180,E1 7521.651,E2 7521.651} C_VEL
LIN {X 0,Y 608.912,Z 923.03,A -85,B 0,C 180,E1 7526.912,E2 7526.912} C_VEL
LIN {X 0,Y 608.97,Z 923.03,A -85,B 0,C 180,E1 7531.872,E2 7531.872} C_VEL
LIN {X 0,Y 609.095,Z 923.03,A -85,B 0,C 180,E1 7536.644,E2 7536.644} C_VEL
LIN {X 0,Y 608.996,Z 923.03,A -85,B 0,C 180,E1 7541.183,E2 7541.183} C_VEL
LIN {X 0,Y 609.224,Z 923.03,A -85,B 0,C 180,E1 7547.103,E2 7547.103} C_VEL
LIN {X 0,Y 609.457,Z 923.03,A -85,B 0,C 180,E1 7552.699,E2 7552.699} C_VEL
LIN {X 0,Y 609.434,Z 923.476,A -85,B 0,C 180,E1 7555.023,E2 7555.023} C_VEL
LIN {X 0,Y 613.83,Z 949.253,A -85,B 0,C 180,E1 7555.47,E2 7555.47} C_VEL
LIN {X 0,Y 613.792,Z 983.938,A -85,B 0,C 180,E1 7556.066,E2 7556.066} C_VEL
LIN {X 0,Y 613.281,Z 1012.694,A -85,B 0,C 180,E1 7557.115,E2 7557.115} C_VEL
LIN {X 0,Y 612.614,Z 1038.233,A -85,B 0,C 180,E1 7558.667,E2 7558.667} C_VEL
LIN {X 0,Y 611.982,Z 1059.146,A -85,B 0,C 180,E1 7560.567,E2 7560.567} C_VEL
LIN {X 0,Y 611.354,Z 1075.944,A -85,B 0,C 180,E1 7562.835,E2 7562.835} C_VEL
LIN {X 0,Y 610.813,Z 1087.678,A -85,B 0,C 180,E1 7565.325,E2 7565.325} C_VEL
LIN {X 0,Y 610.574,Z 1094.316,A -85,B 0,C 180,E1 7568.078,E2 7568.078} C_VEL
LIN {X 0,Y 610.508,Z 1095.452,A -85,B 0,C 180,E1 7569.979,E2 7569.979} C_VEL
LIN {X 0,Y 610.584,Z 1093.085,A -85,B 0,C 180,E1 7572.321,E2 7572.321} C_VEL
LIN {X 0,Y 610.787,Z 1086.052,A -85,B 0,C 180,E1 7574.774,E2 7574.774} C_VEL
LIN {X 0,Y 611.194,Z 1073.436,A -85,B 0,C 180,E1 7577.26,E2 7577.26} C_VEL
LIN {X 0,Y 611.748,Z 1055.978,A -85,B 0,C 180,E1 7579.481,E2 7579.481} C_VEL
LIN {X 0,Y 612.473,Z 1033.258,A -85,B 0,C 180,E1 7581.437,E2 7581.437} C_VEL
LIN {X 0,Y 613.185,Z 1006.915,A -85,B 0,C 180,E1 7582.931,E2 7582.931} C_VEL
LIN {X 0,Y 613.608,Z 977.971,A -85,B 0,C 180,E1 7583.916,E2 7583.916} C_VEL
LIN {X 0,Y 613.054,Z 941.178,A -85,B 0,C 180,E1 7584.497,E2 7584.497} C_VEL
LIN {X 0,Y 609.271,Z 923.03,A -85,B 0,C 180,E1 7584.846,E2 7584.846} C_VEL
LIN {X 0,Y 608.884,Z 923.03,A -85,B 0,C 180,E1 7589.761,E2 7589.761} C_VEL
LIN {X 0,Y 608.849,Z 923.03,A -85,B 0,C 180,E1 7594.999,E2 7594.999} C_VEL
LIN {X 0,Y 608.799,Z 923.03,A -85,B 0,C 180,E1 7600.193,E2 7600.193} C_VEL
LIN {X 0,Y 608.79,Z 923.03,A -85,B 0,C 180,E1 7606.042,E2 7606.042} C_VEL
LIN {X 0,Y 608.87,Z 923.03,A -85,B 0,C 180,E1 7611.639,E2 7611.639} C_VEL
LIN {X 0,Y 608.89,Z 923.03,A -85,B 0,C 180,E1 7617.545,E2 7617.545} C_VEL
LIN {X 0,Y 609.107,Z 923.03,A -85,B 0,C 180,E1 7623.466,E2 7623.466} C_VEL
LIN {X 0,Y 609.117,Z 923.03,A -85,B 0,C 180,E1 7628.142,E2 7628.142} C_VEL
LIN {X 0,Y 609.247,Z 923.03,A -85,B 0,C 180,E1 7632.673,E2 7632.673} C_VEL
LIN {X 0,Y 609.325,Z 923.03,A -85,B 0,C 180,E1 7638.545,E2 7638.545} C_VEL
LIN {X 0,Y 609.497,Z 923.03,A -85,B 0,C 180,E1 7644.297,E2 7644.297} C_VEL
LIN {X 0,Y 609.629,Z 923.03,A -85,B 0,C 180,E1 7648.567,E2 7648.567} C_VEL
LIN {X 0,Y 609.563,Z 923.03,A -85,B 0,C 180,E1 7652.829,E2 7652.829} C_VEL
LIN {X 0,Y 609.459,Z 923.03,A -85,B 0,C 180,E1 7657.347,E2 7657.347} C_VEL
LIN {X 0,Y 609.341,Z 923.03,A -85,B 0,C 180,E1 7662.882,E2 7662.882} C_VEL
LIN {X 0,Y 609.281,Z 923.03,A -85,B 0,C 180,E1 7667.3,E2 7667.3} C_VEL
LIN {X 0,Y 609.131,Z 923.03,A -85,B 0,C 180,E1 7671.83,E2 7671.83} C_VEL
LIN {X 0,Y 609.048,Z 923.03,A -85,B 0,C 180,E1 7676.72,E2 7676.72} C_VEL
LIN {X 0,Y 609.005,Z 923.03,A -85,B 0,C 180,E1 7682.472,E2 7682.472} C_VEL
LIN {X 0,Y 608.86,Z 923.03,A -85,B 0,C 180,E1 7688.33,E2 7688.33} C_VEL
LIN {X 0,Y 608.955,Z 923.03,A -85,B 0,C 180,E1 7693.989,E2 7693.989} C_VEL
LIN {X 0,Y 608.862,Z 923.03,A -85,B 0,C 180,E1 7699.812,E2 7699.812} C_VEL
LIN {X 0,Y 608.812,Z 923.03,A -85,B 0,C 180,E1 7705.187,E2 7705.187} C_VEL
LIN {X 0,Y 609.051,Z 923.03,A -85,B 0,C 180,E1 7711.063,E2 7711.063} C_VEL
LIN {X 0,Y 609.122,Z 923.03,A -85,B 0,C 180,E1 7711.491,E2 7711.491} C_VEL
LIN {X 0,Y 622.373,Z 963.459,A -85,B 0,C 180,E1 7713.003,E2 7713.003} C_VEL
LIN {X 0,Y 620.355,Z 1002.328,A -85,B 0,C 180,E1 7714.369,E2 7714.369} C_VEL
LIN {X 0,Y 618.181,Z 1038.036,A -85,B 0,C 180,E1 7716.2,E2 7716.2} C_VEL
LIN {X 0,Y 615.739,Z 1071.85,A -85,B 0,C 180,E1 7718.562,E2 7718.562} C_VEL
LIN {X 0,Y 613.577,Z 1101.464,A -85,B 0,C 180,E1 7721.326,E2 7721.326} C_VEL
LIN {X 0,Y 611.953,Z 1126.374,A -85,B 0,C 180,E1 7724.419,E2 7724.419} C_VEL
LIN {X 0,Y 610.734,Z 1146.758,A -85,B 0,C 180,E1 7727.849,E2 7727.849} C_VEL
LIN {X 0,Y 610.142,Z 1161.719,A -85,B 0,C 180,E1 7731.453,E2 7731.453} C_VEL
LIN {X 0,Y 609.879,Z 1171.019,A -85,B 0,C 180,E1 7735.024,E2 7735.024} C_VEL
LIN {X 0,Y 609.769,Z 1175.274,A -85,B 0,C 180,E1 7738.578,E2 7738.578} C_VEL
LIN {X 0,Y 609.773,Z 1175.217,A -85,B 0,C 180,E1 7741.418,E2 7741.418} C_VEL
LIN {X 0,Y 609.906,Z 1170.895,A -85,B 0,C 180,E1 7744.973,E2 7744.973} C_VEL
LIN {X 0,Y 610.13,Z 1161.516,A -85,B 0,C 180,E1 7748.544,E2 7748.544} C_VEL
LIN {X 0,Y 610.744,Z 1146.463,A -85,B 0,C 180,E1 7752.147,E2 7752.147} C_VEL
LIN {X 0,Y 611.925,Z 1125.992,A -85,B 0,C 180,E1 7755.563,E2 7755.563} C_VEL
LIN {X 0,Y 613.612,Z 1100.57,A -85,B 0,C 180,E1 7758.67,E2 7758.67} C_VEL
LIN {X 0,Y 615.628,Z 1071.998,A -85,B 0,C 180,E1 7761.299,E2 7761.299} C_VEL
LIN {X 0,Y 617.927,Z 1038.471,A -85,B 0,C 180,E1 7763.608,E2 7763.608} C_VEL
LIN {X 0,Y 619.916,Z 1003.189,A -85,B 0,C 180,E1 7765.39,E2 7765.39} C_VEL
LIN {X 0,Y 621.564,Z 966.179,A -85,B 0,C 180,E1 7766.689,E2 7766.689} C_VEL
LIN {X 0,Y 619.655,Z 956.796,A -85,B 0,C 180,E1 7767.03,E2 7767.03} C_VEL
LIN {X 0,Y 609.109,Z 923.03,A -85,B 0,C 180,E1 7768.223,E2 7768.223} C_VEL
LIN {X 0,Y 609.007,Z 923.03,A -85,B 0,C 180,E1 7773.083,E2 7773.083} C_VEL
LIN {X 0,Y 608.786,Z 923.03,A -85,B 0,C 180,E1 7777.668,E2 7777.668} C_VEL
LIN {X 0,Y 604.817,Z 923.03,A -85,B 0,C 180,E1 7779.269,E2 7779.269} C_VEL
LIN {X 0,Y 600.837,Z 923.03,A -85,B 0,C 180,E1 7780.89,E2 7780.89} C_VEL
LIN {X 0,Y 600.8,Z 923.03,A -85,B 0,C 180,E1 7786.833,E2 7786.833} C_VEL
LIN {X 0,Y 600.976,Z 923.03,A -85,B 0,C 180,E1 7792.902,E2 7792.902} C_VEL
LIN {X 0,Y 601.01,Z 923.03,A -85,B 0,C 180,E1 7798.74,E2 7798.74} C_VEL
LIN {X 0,Y 601.051,Z 923.03,A -85,B 0,C 180,E1 7800.666,E2 7800.666} C_VEL
LIN {X 0,Y 615.219,Z 966.833,A -85,B 0,C 180,E1 7801.961,E2 7801.961} C_VEL
LIN {X 0,Y 613.965,Z 1011.28,A -85,B 0,C 180,E1 7802.784,E2 7802.784} C_VEL
LIN {X 0,Y 612.084,Z 1052.394,A -85,B 0,C 180,E1 7804.139,E2 7804.139} C_VEL
LIN {X 0,Y 609.986,Z 1088.781,A -85,B 0,C 180,E1 7805.891,E2 7805.891} C_VEL
LIN {X 0,Y 607.804,Z 1122.814,A -85,B 0,C 180,E1 7808.12,E2 7808.12} C_VEL
LIN {X 0,Y 605.742,Z 1152.788,A -85,B 0,C 180,E1 7810.714,E2 7810.714} C_VEL
LIN {X 0,Y 604.125,Z 1178.786,A -85,B 0,C 180,E1 7813.671,E2 7813.671} C_VEL
LIN {X 0,Y 602.936,Z 1200.546,A -85,B 0,C 180,E1 7816.978,E2 7816.978} C_VEL
LIN {X 0,Y 602.325,Z 1216.226,A -85,B 0,C 180,E1 7820.264,E2 7820.264} C_VEL
LIN {X 0,Y 602.052,Z 1226.843,A -85,B 0,C 180,E1 7823.528,E2 7823.528} C_VEL
LIN {X 0,Y 601.947,Z 1233.399,A -85,B 0,C 180,E1 7827.135,E2 7827.135} C_VEL
LIN {X 0,Y 601.922,Z 1235.042,A -85,B 0,C 180,E1 7830.013,E2 7830.013} C_VEL
LIN {X 0,Y 601.933,Z 1232.517,A -85,B 0,C 180,E1 7833.611,E2 7833.611} C_VEL
LIN {X 0,Y 602.077,Z 1224.894,A -85,B 0,C 180,E1 7837.221,E2 7837.221} C_VEL
LIN {X 0,Y 602.488,Z 1211.737,A -85,B 0,C 180,E1 7840.854,E2 7840.854} C_VEL
LIN {X 0,Y 603.444,Z 1192.196,A -85,B 0,C 180,E1 7844.514,E2 7844.514} C_VEL
LIN {X 0,Y 605.055,Z 1166.617,A -85,B 0,C 180,E1 7847.955,E2 7847.955} C_VEL
LIN {X 0,Y 607.11,Z 1137.58,A -85,B 0,C 180,E1 7850.876,E2 7850.876} C_VEL
LIN {X 0,Y 609.532,Z 1104.613,A -85,B 0,C 180,E1 7853.381,E2 7853.381} C_VEL
LIN {X 0,Y 611.992,Z 1069.29,A -85,B 0,C 180,E1 7855.375,E2 7855.375} C_VEL
LIN {X 0,Y 614.243,Z 1031.553,A -85,B 0,C 180,E1 7856.886,E2 7856.886} C_VEL
LIN {X 0,Y 615.864,Z 992.283,A -85,B 0,C 180,E1 7857.892,E2 7857.892} C_VEL
LIN {X 0,Y 615.881,Z 963.739,A -85,B 0,C 180,E1 7858.348,E2 7858.348} C_VEL
LIN {X 0,Y 601.078,Z 923.03,A -85,B 0,C 180,E1 7859.641,E2 7859.641} C_VEL
LIN {X 0,Y 600.986,Z 923.03,A -85,B 0,C 180,E1 7865.343,E2 7865.343} C_VEL
